C01796=1071.696,311.652,-94.387,174.617,30.497,155.487
C01797=1071.686,311.264,-94.337,174.612,30.490,155.486
C01798=1071.676,310.875,-94.286,174.607,30.483,155.484
C01799=1071.666,310.487,-94.236,174.603,30.476,155.483
C01800=1071.656,310.099,-94.186,174.597,30.469,155.482
C01801=1071.650,309.851,-94.154,174.595,30.465,155.481
C01802=1071.644,309.604,-94.121,174.592,30.460,155.480
C01803=1071.638,309.356,-94.089,174.589,30.456,155.480
C01804=1071.632,309.108,-94.057,174.586,30.451,155.479
C01805=1071.626,308.860,-94.025,174.582,30.447,155.478
C01806=1071.619,308.612,-93.993,174.580,30.443,155.477
C01807=1071.613,308.365,-93.960,174.577,30.439,155.477
C01808=1071.608,308.117,-93.929,174.573,30.434,155.476
C01809=1071.602,307.869,-93.897,174.571,30.430,155.475
C01810=1071.596,307.621,-93.865,174.567,30.425,155.474
C01811=1071.589,307.374,-93.833,174.565,30.421,155.473
C01812=1071.583,307.126,-93.801,174.562,30.417,155.473
C01813=1071.577,306.878,-93.769,174.558,30.412,155.472
C01814=1071.571,306.630,-93.737,174.556,30.408,155.471
C01815=1071.564,306.382,-93.705,174.552,30.403,155.470
C01816=1071.559,306.135,-93.673,174.550,30.399,155.470
C01817=1071.553,305.887,-93.641,174.547,30.395,155.469
C01818=1071.547,305.638,-93.609,174.543,30.390,155.468
C01819=1071.540,305.390,-93.578,174.541,30.386,155.467
C01820=1071.535,305.143,-93.546,174.538,30.382,155.467
C01821=1071.529,304.895,-93.513,174.535,30.377,155.466
C01822=1071.523,304.647,-93.481,174.532,30.373,155.465
C01823=1071.516,304.400,-93.450,174.529,30.368,155.464
C01824=1071.510,304.152,-93.418,174.526,30.364,155.463
C01825=1071.503,303.847,-93.379,174.522,30.359,155.463
C01826=1071.496,303.543,-93.340,174.519,30.354,155.462
C01827=1071.488,303.240,-93.301,174.515,30.348,155.461
C01828=1071.481,302.936,-93.263,174.512,30.343,155.460
C01829=1071.475,302.687,-93.231,174.508,30.338,155.459
C01830=1071.469,302.439,-93.199,174.506,30.334,155.458
C01831=1071.463,302.192,-93.167,174.503,30.330,155.457
C01832=1071.457,301.944,-93.135,174.499,30.325,155.457
C01833=1071.452,301.696,-93.104,174.497,30.321,155.456
C01834=1071.445,301.448,-93.072,174.494,30.317,155.455
C01835=1071.440,301.201,-93.041,174.492,30.313,155.454
C01836=1071.434,300.952,-93.009,174.488,30.308,155.454
C01837=1071.427,300.704,-92.978,174.485,30.304,155.453
C01838=1071.422,300.457,-92.946,174.483,30.299,155.452
C01839=1071.416,300.208,-92.914,174.479,30.295,155.451
C01840=1071.410,299.961,-92.883,174.477,30.291,155.451
C01841=1071.404,299.713,-92.851,174.474,30.287,155.450
C01842=1071.399,299.465,-92.820,174.470,30.282,155.449
C01843=1071.392,299.217,-92.789,174.468,30.278,155.448
C01844=1071.387,298.969,-92.757,174.465,30.273,155.448
C01845=1071.380,298.721,-92.726,174.463,30.270,155.447
C01846=1071.375,298.473,-92.695,174.459,30.265,155.446
C01847=1071.369,298.225,-92.663,174.456,30.261,155.445
C01848=1071.363,297.978,-92.632,174.454,30.256,155.445
C01849=1071.357,297.729,-92.600,174.450,30.252,155.444
C01850=1071.352,297.482,-92.569,174.448,30.248,155.443
C01851=1071.345,297.234,-92.537,174.445,30.243,155.442
C01852=1071.339,296.986,-92.507,174.442,30.239,155.442
C01853=1071.333,296.738,-92.475,174.439,30.235,155.441
C01854=1071.327,296.490,-92.444,174.436,30.231,155.440
C01855=1071.321,296.242,-92.412,174.434,30.226,155.439
C01856=1071.316,295.994,-92.382,174.431,30.222,155.439
C01857=1071.309,295.746,-92.351,174.427,30.218,155.438
C01858=1071.304,295.498,-92.319,174.425,30.214,155.437
C01859=1071.297,295.250,-92.288,174.422,30.210,155.436
C01860=1071.291,295.002,-92.258,174.420,30.205,155.436
C01861=1071.285,294.754,-92.227,174.416,30.201,155.435
C01862=1071.279,294.506,-92.196,174.414,30.197,155.434
C01863=1071.273,294.259,-92.165,174.411,30.193,155.434
C01864=1071.267,294.010,-92.134,174.408,30.189,155.433
C01865=1071.262,293.763,-92.102,174.405,30.184,155.432
C01866=1071.255,293.514,-92.071,174.402,30.180,155.431
C01867=1071.249,293.266,-92.041,174.400,30.176,155.431
C01868=1071.243,293.019,-92.010,174.397,30.172,155.430
C01869=1071.237,292.771,-91.979,174.393,30.167,155.429
C01870=1071.231,292.522,-91.948,174.391,30.164,155.429
C01871=1071.225,292.275,-91.917,174.388,30.159,155.428
C01872=1071.219,292.027,-91.887,174.386,30.155,155.427
C01873=1071.213,291.778,-91.856,174.382,30.151,155.426
C01874=1071.208,291.530,-91.825,174.379,30.147,155.426
C01875=1071.202,291.283,-91.794,174.377,30.143,155.425
C01876=1071.195,291.034,-91.763,174.374,30.139,155.424
C01877=1071.190,290.820,-91.736,174.372,30.135,155.424
C01878=1071.185,290.605,-91.709,174.369,30.131,155.423
C01879=1071.180,290.390,-91.684,174.366,30.128,155.422
C01880=1071.174,290.175,-91.657,174.365,30.124,155.422
C01881=1071.169,289.960,-91.630,174.362,30.120,155.421
C01882=1071.164,289.745,-91.603,174.359,30.117,155.420
C01883=1071.159,289.530,-91.577,174.357,30.113,155.420
C01884=1071.154,289.315,-91.551,174.355,30.109,155.419
C01885=1071.148,289.068,-91.520,174.352,30.105,155.419
C01886=1071.142,288.819,-91.489,174.349,30.101,155.418
C01887=1071.136,288.571,-91.459,174.346,30.097,155.417
C01888=1071.129,288.323,-91.428,174.344,30.093,155.416
C01889=1071.124,288.076,-91.397,174.341,30.089,155.416
C01890=1071.118,287.828,-91.367,174.338,30.085,155.415
C01891=1071.111,287.579,-91.336,174.335,30.080,155.414
C01892=1071.106,287.331,-91.306,174.332,30.077,155.414
C01893=1071.099,287.084,-91.276,174.330,30.073,155.413
C01894=1071.093,286.835,-91.245,174.327,30.068,155.412
C01895=1071.087,286.587,-91.216,174.324,30.064,155.411
C01896=1071.081,286.339,-91.185,174.321,30.060,155.411
C01897=1071.075,286.091,-91.155,174.318,30.056,155.410
C01898=1071.069,285.843,-91.124,174.316,30.052,155.409
C01899=1071.063,285.595,-91.094,174.313,30.048,155.409
C01900=1071.057,285.347,-91.064,174.311,30.044,155.408
C01901=1071.052,285.099,-91.033,174.307,30.040,155.407
C01902=1071.045,284.851,-91.003,174.305,30.035,155.407
C01903=1071.039,284.603,-90.972,174.302,30.032,155.406
C01904=1071.034,284.354,-90.943,174.299,30.027,155.405
C01905=1071.028,284.107,-90.912,174.297,30.023,155.404
C01906=1071.022,283.858,-90.882,174.294,30.019,155.404
C01907=1071.015,283.611,-90.852,174.291,30.015,155.403
C01908=1071.009,283.363,-90.821,174.288,30.011,155.402
C01909=1071.004,283.114,-90.792,174.286,30.007,155.402
C01910=1070.998,282.867,-90.761,174.283,30.003,155.401
C01911=1070.991,282.618,-90.731,174.280,29.999,155.400
C01912=1070.986,282.370,-90.701,174.278,29.994,155.399
C01913=1070.980,282.122,-90.671,174.275,29.991,155.399
C01914=1070.974,281.874,-90.640,174.272,29.986,155.398
C01915=1070.969,281.625,-90.611,174.269,29.982,155.397
C01916=1070.962,281.378,-90.581,174.266,29.978,155.397
C01917=1070.956,281.129,-90.550,174.264,29.974,155.396
C01918=1070.950,280.881,-90.521,174.261,29.970,155.395
C01919=1070.945,280.633,-90.490,174.259,29.966,155.395
C01920=1070.939,280.385,-90.460,174.256,29.962,155.394
C01921=1070.932,280.137,-90.431,174.254,29.958,155.393
C01922=1070.927,279.889,-90.401,174.251,29.954,155.393
C01923=1070.921,279.641,-90.371,174.248,29.949,155.392
C01924=1070.914,279.393,-90.341,174.245,29.945,155.391
C01925=1070.908,279.144,-90.311,174.242,29.942,155.391
C01926=1070.903,278.896,-90.281,174.240,29.937,155.390
C01927=1070.896,278.648,-90.252,174.237,29.933,155.389
C01928=1070.891,278.401,-90.221,174.235,29.929,155.388
C01929=1070.885,278.152,-90.192,174.232,29.926,155.388
C01930=1070.879,277.904,-90.163,174.229,29.921,155.387
C01931=1070.873,277.656,-90.132,174.227,29.917,155.386
C01932=1070.867,277.408,-90.103,174.223,29.913,155.386
C01933=1070.857,276.988,-90.052,174.219,29.906,155.384
C01934=1070.846,276.569,-90.002,174.215,29.899,155.383
C01935=1070.836,276.149,-89.952,174.210,29.893,155.382
C01936=1070.826,275.729,-89.902,174.206,29.886,155.381
C01937=1070.821,275.481,-89.872,174.204,29.882,155.380
C01938=1070.814,275.233,-89.843,174.200,29.878,155.380
C01939=1070.809,274.985,-89.813,174.198,29.873,155.379
C01940=1070.803,274.737,-89.784,174.195,29.869,155.378
C01941=1070.797,274.489,-89.754,174.192,29.866,155.378
C01942=1070.790,274.241,-89.725,174.190,29.862,155.377
C01943=1070.785,273.992,-89.695,174.187,29.857,155.376
C01944=1070.779,273.744,-89.666,174.185,29.853,155.376
C01945=1070.773,273.496,-89.636,174.182,29.849,155.375
C01946=1070.768,273.247,-89.607,174.180,29.846,155.374
C01947=1070.761,273.000,-89.577,174.177,29.841,155.373
C01948=1070.755,272.752,-89.548,174.174,29.837,155.373
C01949=1070.749,272.503,-89.518,174.172,29.833,155.372
C01950=1070.743,272.255,-89.489,174.169,29.829,155.371
C01951=1070.738,272.007,-89.459,174.167,29.826,155.371
C01952=1070.731,271.758,-89.430,174.164,29.821,155.370
C01953=1070.725,271.510,-89.401,174.162,29.817,155.369
C01954=1070.720,271.262,-89.372,174.159,29.813,155.369
C01955=1070.713,271.014,-89.343,174.156,29.809,155.368
C01956=1070.708,270.765,-89.313,174.153,29.805,155.367
C01957=1070.702,270.517,-89.284,174.150,29.801,155.367
C01958=1070.696,270.270,-89.255,174.148,29.797,155.366
C01959=1070.690,270.021,-89.226,174.145,29.793,155.365
C01960=1070.684,269.773,-89.197,174.143,29.789,155.365
C01961=1070.678,269.525,-89.168,174.140,29.785,155.364
C01962=1070.672,269.277,-89.138,174.138,29.781,155.363
C01963=1070.666,269.028,-89.109,174.135,29.777,155.363
C01964=1070.660,268.780,-89.080,174.132,29.773,155.362
C01965=1070.654,268.532,-89.050,174.130,29.769,155.361
C01966=1070.648,268.284,-89.021,174.127,29.765,155.361
C01967=1070.642,268.035,-88.993,174.125,29.761,155.360
C01968=1070.636,267.787,-88.964,174.122,29.757,155.359
C01969=1070.630,267.539,-88.935,174.120,29.753,155.359
C01970=1070.625,267.291,-88.906,174.117,29.749,155.358
C01971=1070.619,267.043,-88.877,174.115,29.745,155.357
C01972=1070.613,266.794,-88.848,174.112,29.741,155.357
C01973=1070.606,266.546,-88.819,174.109,29.738,155.356
C01974=1070.601,266.297,-88.790,174.107,29.733,155.355
C01975=1070.595,266.049,-88.761,174.104,29.729,155.355
C01976=1070.589,265.801,-88.732,174.102,29.725,155.354
C01977=1070.583,265.553,-88.704,174.099,29.721,155.353
C01978=1070.577,265.305,-88.674,174.097,29.717,155.353
C01979=1070.571,265.057,-88.645,174.094,29.713,155.352
C01980=1070.565,264.808,-88.617,174.092,29.709,155.351
C01981=1070.559,264.560,-88.587,174.089,29.705,155.351
C01982=1070.553,264.312,-88.558,174.087,29.701,155.350
C01983=1070.547,264.064,-88.530,174.084,29.697,155.349
C01984=1070.541,263.815,-88.501,174.081,29.694,155.349
C01985=1070.531,263.399,-88.453,174.077,29.686,155.347
C01986=1070.521,262.982,-88.406,174.073,29.680,155.346
C01987=1070.511,262.566,-88.357,174.069,29.673,155.345
C01988=1070.501,262.150,-88.309,174.064,29.667,155.344
C01989=1070.495,261.901,-88.281,174.062,29.663,155.343
C01990=1070.489,261.654,-88.252,174.059,29.659,155.343
C01991=1070.483,261.405,-88.224,174.057,29.655,155.342
C01992=1070.477,261.157,-88.195,174.054,29.651,155.342
C01993=1070.470,260.909,-88.167,174.052,29.647,155.341
C01994=1070.464,260.661,-88.138,174.049,29.643,155.340
C01995=1070.458,260.412,-88.110,174.047,29.640,155.340
C01996=1070.453,260.164,-88.082,174.044,29.636,155.339
C01997=1070.446,259.916,-88.053,174.042,29.632,155.338
C01998=1070.440,259.667,-88.025,174.040,29.628,155.338
C01999=1070.434,259.419,-87.996,174.037,29.624,155.337
C02000=1070.428,259.171,-87.968,174.035,29.620,155.336
C02001=1070.422,258.922,-87.940,174.032,29.616,155.336
C02002=1070.416,258.674,-87.911,174.030,29.612,155.335
C02003=1070.410,258.425,-87.883,174.027,29.608,155.334
C02004=1070.405,258.177,-87.855,174.025,29.604,155.334
C02005=1070.399,257.929,-87.826,174.022,29.601,155.333
C02006=1070.392,257.681,-87.798,174.019,29.597,155.332
C02007=1070.386,257.433,-87.770,174.017,29.592,155.332
C02008=1070.380,257.184,-87.741,174.014,29.588,155.331
C02009=1070.374,256.935,-87.713,174.012,29.584,155.330
C02010=1070.369,256.688,-87.684,174.009,29.580,155.330
C02011=1070.362,256.439,-87.657,174.007,29.576,155.329
C02012=1070.356,256.191,-87.628,174.004,29.573,155.328
C02013=1070.351,255.943,-87.600,174.003,29.569,155.328
C02014=1070.345,255.694,-87.572,174.000,29.565,155.327
C02015=1070.339,255.445,-87.544,173.998,29.561,155.326
C02016=1070.333,255.198,-87.516,173.995,29.557,155.326
C02017=1070.327,254.949,-87.487,173.993,29.553,155.325
C02018=1070.321,254.700,-87.459,173.990,29.549,155.325
C02019=1070.315,254.452,-87.431,173.988,29.545,155.324
C02020=1070.309,254.204,-87.403,173.985,29.541,155.323
C02021=1070.303,253.956,-87.375,173.982,29.537,155.322
C02022=1070.297,253.707,-87.347,173.980,29.533,155.322
C02023=1070.291,253.458,-87.319,173.978,29.529,155.321
C02024=1070.285,253.211,-87.291,173.976,29.525,155.320
C02025=1070.279,252.962,-87.263,173.973,29.521,155.320
C02026=1070.274,252.714,-87.235,173.971,29.517,155.319
C02027=1070.268,252.465,-87.207,173.968,29.513,155.318
C02028=1070.261,252.217,-87.179,173.966,29.509,155.318
C02029=1070.256,251.969,-87.151,173.963,29.505,155.317
C02030=1070.250,251.720,-87.123,173.961,29.501,155.316
C02031=1070.245,251.472,-87.095,173.958,29.497,155.316
C02032=1070.238,251.223,-87.067,173.957,29.494,155.315
C02033=1070.233,250.975,-87.039,173.954,29.490,155.315
C02034=1070.227,250.726,-87.011,173.952,29.485,155.314
C02035=1070.221,250.478,-86.983,173.949,29.481,155.313
C02036=1070.215,250.229,-86.956,173.947,29.477,155.312
C02037=1070.205,249.811,-86.909,173.942,29.471,155.311
C02038=1070.196,249.392,-86.862,173.938,29.464,155.310
C02039=1070.186,248.974,-86.815,173.935,29.457,155.309
C02040=1070.176,248.555,-86.768,173.931,29.451,155.308
C02041=1070.170,248.307,-86.740,173.928,29.446,155.307
C02042=1070.165,248.059,-86.712,173.926,29.442,155.307
C02043=1070.159,247.810,-86.685,173.923,29.438,155.306
C02044=1070.153,247.562,-86.657,173.921,29.434,155.305
C02045=1070.147,247.313,-86.629,173.919,29.431,155.305
C02046=1070.142,247.065,-86.602,173.917,29.426,155.304
C02047=1070.135,246.816,-86.574,173.914,29.422,155.303
C02048=1070.130,246.568,-86.546,173.912,29.418,155.303
C02049=1070.124,246.320,-86.519,173.909,29.414,155.302
C02050=1070.118,246.071,-86.491,173.907,29.410,155.301
C02051=1070.112,245.823,-86.464,173.905,29.407,155.301
C02052=1070.107,245.574,-86.436,173.902,29.403,155.300
C02053=1070.101,245.326,-86.409,173.900,29.399,155.299
C02054=1070.094,245.078,-86.381,173.897,29.395,155.299
C02055=1070.089,244.829,-86.354,173.895,29.390,155.298
C02056=1070.083,244.581,-86.326,173.892,29.386,155.297
C02057=1070.077,244.332,-86.299,173.891,29.383,155.297
C02058=1070.071,244.084,-86.271,173.888,29.379,155.296
C02059=1070.065,243.835,-86.244,173.886,29.375,155.295
C02060=1070.059,243.587,-86.216,173.883,29.371,155.295
C02061=1070.054,243.339,-86.189,173.881,29.367,155.294
C02062=1070.048,243.090,-86.161,173.879,29.363,155.293
C02063=1070.042,242.842,-86.135,173.877,29.359,155.293
C02064=1070.037,242.594,-86.107,173.874,29.355,155.292
C02065=1070.030,242.345,-86.080,173.872,29.351,155.291
C02066=1070.024,242.097,-86.052,173.869,29.347,155.291
C02067=1070.018,241.847,-86.025,173.868,29.343,155.290
C02068=1070.013,241.599,-85.998,173.865,29.339,155.289
C02069=1070.006,241.351,-85.970,173.863,29.335,155.289
C02070=1070.000,241.102,-85.944,173.860,29.331,155.288
C02071=1069.994,240.854,-85.917,173.858,29.327,155.287
C02072=1069.989,240.605,-85.889,173.856,29.324,155.287
C02073=1069.983,240.357,-85.862,173.854,29.320,155.286
C02074=1069.977,240.108,-85.836,173.851,29.316,155.285
C02075=1069.970,239.860,-85.808,173.849,29.312,155.285
C02076=1069.965,239.611,-85.781,173.846,29.308,155.284
C02077=1069.959,239.363,-85.754,173.845,29.304,155.284
C02078=1069.953,239.115,-85.726,173.842,29.300,155.283
C02079=1069.947,238.866,-85.700,173.840,29.296,155.282
C02080=1069.941,238.618,-85.673,173.837,29.292,155.281
C02081=1069.935,238.369,-85.646,173.835,29.288,155.281
C02082=1069.930,238.120,-85.619,173.833,29.284,155.280
C02083=1069.924,237.872,-85.591,173.831,29.280,155.280
C02084=1069.917,237.623,-85.564,173.828,29.276,155.279
C02085=1069.912,237.375,-85.538,173.826,29.272,155.278
C02086=1069.906,237.127,-85.511,173.824,29.268,155.278
C02087=1069.900,236.878,-85.484,173.822,29.264,155.277
C02088=1069.894,236.629,-85.457,173.819,29.260,155.276
C02089=1069.889,236.417,-85.434,173.818,29.257,155.276
C02090=1069.884,236.205,-85.411,173.815,29.253,155.275
C02091=1069.879,235.992,-85.388,173.813,29.250,155.275
C02092=1069.875,235.780,-85.365,173.812,29.247,155.274
C02093=1069.869,235.567,-85.342,173.809,29.243,155.273
C02094=1069.864,235.354,-85.319,173.808,29.240,155.273
C02095=1069.859,235.142,-85.296,173.806,29.236,155.272
C02096=1069.854,234.929,-85.273,173.804,29.233,155.272
C02097=1069.848,234.681,-85.246,173.801,29.229,155.271
C02098=1069.842,234.432,-85.219,173.800,29.225,155.270
C02099=1069.836,234.184,-85.192,173.797,29.221,155.270
C02100=1069.830,233.936,-85.166,173.795,29.217,155.269
C02101=1069.824,233.687,-85.139,173.792,29.213,155.268
C02102=1069.819,233.439,-85.112,173.791,29.209,155.268
C02103=1069.813,233.189,-85.086,173.788,29.205,155.267
C02104=1069.807,232.941,-85.060,173.786,29.201,155.266
C02105=1069.801,232.693,-85.033,173.783,29.197,155.266
C02106=1069.795,232.444,-85.006,173.782,29.193,155.265
C02107=1069.790,232.196,-84.980,173.779,29.189,155.265
C02108=1069.783,231.947,-84.953,173.777,29.185,155.264
C02109=1069.777,231.698,-84.926,173.775,29.181,155.263
C02110=1069.772,231.450,-84.899,173.773,29.177,155.262
C02111=1069.766,231.202,-84.873,173.770,29.173,155.262
C02112=1069.760,230.953,-84.846,173.768,29.169,155.261
C02113=1069.755,230.704,-84.820,173.766,29.166,155.260
C02114=1069.749,230.456,-84.793,173.764,29.162,155.260
C02115=1069.743,230.208,-84.767,173.761,29.158,155.259
C02116=1069.737,229.959,-84.740,173.760,29.154,155.259
C02117=1069.730,229.711,-84.714,173.757,29.149,155.258
C02118=1069.725,229.462,-84.688,173.755,29.145,155.257
C02119=1069.719,229.213,-84.661,173.752,29.141,155.257
C02120=1069.713,228.965,-84.634,173.751,29.138,155.256
C02121=1069.707,228.717,-84.608,173.748,29.134,155.255
C02122=1069.701,228.467,-84.582,173.746,29.130,155.255
C02123=1069.695,228.219,-84.555,173.744,29.126,155.254
C02124=1069.689,227.970,-84.529,173.742,29.122,155.253
C02125=1069.683,227.722,-84.503,173.739,29.118,155.253
C02126=1069.677,227.473,-84.477,173.737,29.114,155.252
C02127=1069.671,227.225,-84.450,173.735,29.110,155.251
C02128=1069.666,226.976,-84.424,173.733,29.106,155.251
C02129=1069.659,226.728,-84.398,173.730,29.102,155.250
C02130=1069.654,226.480,-84.372,173.729,29.098,155.249
C02131=1069.647,226.230,-84.345,173.726,29.094,155.249
C02132=1069.642,225.982,-84.319,173.724,29.090,155.248
C02133=1069.635,225.733,-84.293,173.722,29.086,155.247
C02134=1069.630,225.485,-84.267,173.720,29.082,155.247
C02135=1069.624,225.236,-84.241,173.718,29.078,155.246
C02136=1069.618,224.988,-84.215,173.716,29.074,155.245
C02137=1069.612,224.739,-84.189,173.714,29.070,155.245
C02138=1069.606,224.490,-84.162,173.711,29.066,155.244
C02139=1069.600,224.242,-84.136,173.710,29.062,155.243
C02140=1069.595,223.993,-84.110,173.707,29.058,155.243
C02141=1069.589,223.744,-84.084,173.705,29.054,155.242
C02142=1069.583,223.496,-84.058,173.703,29.050,155.241
C02143=1069.577,223.247,-84.032,173.701,29.046,155.241
C02144=1069.571,222.999,-84.005,173.698,29.042,155.240
C02145=1069.566,222.783,-83.983,173.697,29.039,155.239
C02146=1069.561,222.566,-83.960,173.695,29.035,155.239
C02147=1069.556,222.350,-83.938,173.693,29.031,155.238
C02148=1069.551,222.132,-83.915,173.691,29.028,155.238
C02149=1069.546,221.916,-83.893,173.690,29.025,155.237
C02150=1069.541,221.699,-83.869,173.687,29.021,155.237
C02151=1069.536,221.483,-83.847,173.686,29.018,155.236
C02152=1069.531,221.266,-83.824,173.684,29.015,155.235
C02153=1069.525,221.017,-83.799,173.682,29.010,155.235
C02154=1069.519,220.768,-83.773,173.679,29.006,155.234
C02155=1069.513,220.520,-83.747,173.678,29.002,155.233
C02156=1069.507,220.271,-83.721,173.675,28.998,155.233
C02157=1069.501,220.023,-83.696,173.673,28.994,155.232
C02158=1069.494,219.775,-83.669,173.671,28.991,155.231
C02159=1069.489,219.526,-83.644,173.669,28.987,155.231
C02160=1069.483,219.277,-83.618,173.667,28.983,155.230
C02161=1069.477,219.028,-83.592,173.665,28.979,155.230
C02162=1069.471,218.780,-83.566,173.662,28.975,155.229
C02163=1069.465,218.531,-83.540,173.661,28.970,155.228
C02164=1069.459,218.282,-83.515,173.658,28.966,155.227
C02165=1069.453,218.034,-83.490,173.656,28.962,155.227
C02166=1069.448,217.785,-83.464,173.654,28.959,155.226
C02167=1069.441,217.537,-83.438,173.652,28.955,155.226
C02168=1069.436,217.288,-83.412,173.650,28.951,155.225
C02169=1069.430,217.040,-83.387,173.648,28.947,155.224
C02170=1069.424,216.791,-83.361,173.646,28.942,155.223
C02171=1069.418,216.542,-83.335,173.644,28.939,155.223
C02172=1069.412,216.293,-83.310,173.642,28.935,155.222
C02173=1069.406,216.044,-83.284,173.639,28.931,155.222
C02174=1069.401,215.796,-83.259,173.638,28.927,155.221
C02175=1069.395,215.548,-83.234,173.635,28.922,155.220
C02176=1069.389,215.299,-83.207,173.634,28.919,155.219
C02177=1069.383,215.051,-83.182,173.631,28.914,155.219
C02178=1069.377,214.802,-83.156,173.629,28.910,155.218
C02179=1069.371,214.553,-83.131,173.627,28.907,155.218
C02180=1069.365,214.305,-83.106,173.625,28.902,155.217
C02181=1069.360,214.056,-83.080,173.624,28.898,155.216
C02182=1069.354,213.808,-83.054,173.621,28.894,155.215
C02183=1069.348,213.559,-83.029,173.619,28.890,155.215
C02184=1069.342,213.310,-83.003,173.617,28.886,155.214
C02185=1069.336,213.062,-82.978,173.615,28.882,155.213
C02186=1069.330,212.813,-82.953,173.613,28.878,155.213
C02187=1069.325,212.564,-82.927,173.611,28.874,155.212
C02188=1069.319,212.315,-82.902,173.608,28.870,155.211
C02189=1069.313,212.066,-82.877,173.607,28.866,155.211
C02190=1069.306,211.818,-82.852,173.605,28.862,155.210
C02191=1069.301,211.570,-82.827,173.603,28.858,155.209
C02192=1069.295,211.321,-82.801,173.601,28.854,155.209
C02193=1069.289,211.072,-82.775,173.599,28.850,155.208
C02194=1069.283,210.823,-82.750,173.597,28.846,155.207
C02195=1069.277,210.575,-82.725,173.594,28.842,155.207
C02196=1069.271,210.326,-82.700,173.593,28.838,155.206
C02197=1069.265,210.077,-82.675,173.590,28.834,155.205
C02198=1069.260,209.828,-82.649,173.589,28.830,155.205
C02199=1069.254,209.580,-82.624,173.587,28.826,155.204
C02200=1069.248,209.332,-82.599,173.585,28.822,155.203
C02201=1069.243,209.117,-82.577,173.583,28.818,155.203
C02202=1069.237,208.903,-82.556,173.581,28.815,155.202
C02203=1069.232,208.688,-82.534,173.580,28.811,155.202
C02204=1069.228,208.474,-82.513,173.578,28.808,155.201
C02205=1069.223,208.259,-82.491,173.576,28.804,155.200
C02206=1069.218,208.046,-82.469,173.574,28.801,155.200
C02207=1069.212,207.831,-82.448,173.572,28.798,155.199
C02208=1069.207,207.616,-82.426,173.571,28.794,155.199
C02209=1069.183,206.573,-82.323,173.428,28.722,155.196
C02210=1069.177,206.324,-82.299,173.427,28.718,155.195
C02211=1069.171,206.076,-82.275,173.424,28.715,155.195
C02212=1069.166,205.827,-82.251,173.422,28.712,155.194
C02213=1069.160,205.578,-82.226,173.420,28.709,155.194
C02214=1069.155,205.329,-82.202,173.418,28.706,155.193
C02215=1069.148,205.080,-82.178,173.415,28.703,155.193
C02216=1069.143,204.832,-82.154,173.414,28.700,155.192
C02217=1069.138,204.583,-82.129,173.411,28.697,155.192
C02218=1069.132,204.334,-82.105,173.409,28.693,155.191
C02219=1069.126,204.086,-82.081,173.407,28.690,155.191
C02220=1069.120,203.837,-82.057,173.404,28.687,155.190
C02221=1069.115,203.588,-82.032,173.402,28.684,155.190
C02222=1069.109,203.339,-82.008,173.400,28.681,155.190
C02223=1069.103,203.091,-81.984,173.398,28.678,155.189
C02224=1069.097,202.842,-81.960,173.395,28.675,155.189
C02225=1069.092,202.593,-81.935,173.394,28.672,155.188
C02226=1069.087,202.344,-81.911,173.391,28.669,155.188
C02227=1069.080,202.095,-81.887,173.389,28.665,155.187
C02228=1069.075,201.847,-81.863,173.387,28.662,155.187
C02229=1069.069,201.598,-81.840,173.384,28.660,155.187
C02230=1069.063,201.349,-81.815,173.382,28.656,155.186
C02231=1069.057,201.100,-81.792,173.380,28.653,155.186
C02232=1069.052,200.852,-81.767,173.378,28.650,155.185
C02233=1069.045,200.603,-81.743,173.376,28.647,155.185
C02234=1069.040,200.354,-81.719,173.374,28.644,155.184
C02235=1069.034,200.105,-81.696,173.371,28.641,155.184
C02236=1069.028,199.856,-81.672,173.370,28.638,155.183
C02237=1069.022,199.608,-81.648,173.367,28.635,155.183
C02238=1069.017,199.359,-81.624,173.364,28.632,155.183
C02239=1069.011,199.110,-81.600,173.363,28.629,155.182
C02240=1069.005,198.861,-81.577,173.360,28.626,155.182
C02241=1068.999,198.613,-81.552,173.359,28.623,155.181
C02242=1068.993,198.364,-81.528,173.356,28.620,155.181
C02243=1068.988,198.115,-81.505,173.354,28.617,155.180
C02244=1068.982,197.866,-81.481,173.352,28.614,155.180
C02245=1068.976,197.618,-81.457,173.350,28.611,155.180
C02246=1068.970,197.368,-81.434,173.348,28.608,155.179
C02247=1068.965,197.119,-81.409,173.345,28.605,155.179
C02248=1068.959,196.871,-81.386,173.343,28.602,155.178
C02249=1068.952,196.622,-81.362,173.341,28.599,155.178
C02250=1068.947,196.373,-81.338,173.339,28.596,155.177
C02251=1068.941,196.125,-81.315,173.337,28.593,155.177
C02252=1068.936,195.876,-81.291,173.335,28.590,155.177
C02253=1068.930,195.627,-81.267,173.332,28.587,155.176
C02254=1068.924,195.378,-81.243,173.331,28.584,155.176
C02255=1068.918,195.129,-81.220,173.328,28.581,155.175
C02256=1068.912,194.881,-81.196,173.326,28.578,155.175
C02257=1068.907,194.632,-81.173,173.324,28.575,155.174
C02258=1068.901,194.383,-81.149,173.322,28.572,155.174
C02259=1068.896,194.133,-81.125,173.320,28.569,155.173
C02260=1068.890,193.885,-81.101,173.317,28.566,155.173
C02261=1068.884,193.636,-81.078,173.316,28.563,155.173
C02262=1068.879,193.388,-81.054,173.313,28.560,155.172
C02263=1068.873,193.139,-81.031,173.312,28.557,155.172
C02264=1068.868,192.890,-81.007,173.309,28.554,155.171
C02265=1068.861,192.641,-80.984,173.307,28.551,155.171
C02266=1068.855,192.392,-80.960,173.305,28.548,155.170
C02267=1068.850,192.143,-80.936,173.303,28.545,155.170
C02268=1068.844,191.895,-80.913,173.301,28.542,155.170
C02269=1068.838,191.646,-80.890,173.298,28.538,155.169
C02270=1068.832,191.363,-80.862,173.297,28.536,155.169
C02271=1068.826,191.081,-80.836,173.294,28.532,155.168
C02272=1068.819,190.799,-80.809,173.292,28.529,155.168
C02273=1068.813,190.517,-80.783,173.289,28.525,155.167
C02274=1068.808,190.268,-80.759,173.287,28.522,155.167
C02275=1068.802,190.020,-80.736,173.285,28.519,155.166
C02276=1068.796,189.771,-80.713,173.283,28.516,155.166
C02277=1068.791,189.521,-80.689,173.281,28.513,155.165
C02278=1068.785,189.273,-80.666,173.279,28.510,155.165
C02279=1068.779,189.024,-80.643,173.277,28.507,155.165
C02280=1068.774,188.775,-80.619,173.274,28.504,155.164
C02281=1068.768,188.526,-80.595,173.273,28.501,155.164
C02282=1068.762,188.277,-80.572,173.270,28.498,155.163
C02283=1068.757,188.028,-80.549,173.269,28.495,155.163
C02284=1068.751,187.779,-80.526,173.266,28.492,155.162
C02285=1068.745,187.531,-80.502,173.265,28.489,155.162
C02286=1068.739,187.282,-80.479,173.262,28.486,155.161
C02287=1068.734,187.033,-80.456,173.261,28.483,155.161
C02288=1068.729,186.784,-80.433,173.258,28.480,155.161
C02289=1068.723,186.536,-80.409,173.257,28.477,155.160
C02290=1068.718,186.286,-80.385,173.254,28.474,155.160
C02291=1068.712,186.037,-80.362,173.252,28.471,155.159
C02292=1068.706,185.789,-80.339,173.250,28.468,155.159
C02293=1068.700,185.540,-80.317,173.248,28.465,155.158
C02294=1068.695,185.291,-80.292,173.246,28.462,155.158
C02295=1068.689,185.042,-80.269,173.244,28.459,155.158
C02296=1068.684,184.793,-80.246,173.242,28.456,155.157
C02297=1068.678,184.544,-80.223,173.240,28.453,155.157
C02298=1068.672,184.295,-80.200,173.238,28.450,155.156
C02299=1068.666,184.047,-80.178,173.236,28.448,155.156
C02300=1068.661,183.798,-80.155,173.233,28.445,155.156
C02301=1068.655,183.549,-80.132,173.232,28.442,155.155
C02302=1068.649,183.300,-80.109,173.229,28.439,155.155
C02303=1068.644,183.051,-80.086,173.228,28.436,155.154
C02304=1068.637,182.802,-80.063,173.225,28.433,155.154
C02305=1068.631,182.554,-80.040,173.224,28.430,155.153
C02306=1068.626,182.305,-80.018,173.221,28.427,155.153
C02307=1068.620,182.056,-79.995,173.220,28.424,155.153
C02308=1068.614,181.807,-79.972,173.218,28.422,155.152
C02309=1068.608,181.558,-79.949,173.215,28.419,155.152
C02310=1068.602,181.309,-79.926,173.214,28.416,155.151
C02311=1068.596,181.060,-79.903,173.211,28.413,155.151
C02312=1068.591,180.812,-79.880,173.210,28.410,155.151
C02313=1068.585,180.563,-79.857,173.207,28.407,155.150
C02314=1068.579,180.314,-79.835,173.206,28.405,155.150
C02315=1068.573,180.065,-79.812,173.203,28.402,155.149
C02316=1068.567,179.816,-79.789,173.201,28.399,155.149
C02317=1068.561,179.567,-79.766,173.199,28.396,155.149
C02318=1068.556,179.318,-79.744,173.197,28.393,155.148
C02319=1068.550,179.069,-79.721,173.195,28.390,155.148
C02320=1068.544,178.820,-79.698,173.193,28.387,155.147
C02321=1068.538,178.571,-79.676,173.192,28.385,155.147
C02322=1068.532,178.323,-79.653,173.189,28.382,155.147
C02323=1068.526,178.074,-79.630,173.187,28.379,155.146
C02324=1068.521,177.825,-79.607,173.185,28.376,155.146
C02325=1068.515,177.575,-79.585,173.183,28.373,155.145
C02326=1068.509,177.327,-79.562,173.181,28.370,155.145
C02327=1068.503,177.078,-79.539,173.179,28.367,155.145
C02328=1068.497,176.829,-79.517,173.178,28.364,155.144
C02329=1068.492,176.579,-79.494,173.175,28.361,155.144
C02330=1068.485,176.331,-79.472,173.174,28.359,155.143
C02331=1068.480,176.082,-79.449,173.171,28.356,155.143
C02332=1068.474,175.834,-79.426,173.169,28.353,155.143
C02333=1068.469,175.584,-79.404,173.167,28.350,155.142
C02334=1068.462,175.301,-79.379,173.165,28.347,155.142
C02335=1068.456,175.019,-79.353,173.163,28.344,155.141
C02336=1068.449,174.736,-79.327,173.160,28.340,155.141
C02337=1068.442,174.454,-79.302,173.158,28.337,155.140
C02338=1068.437,174.205,-79.279,173.156,28.334,155.140
C02339=1068.431,173.956,-79.256,173.155,28.331,155.139
C02340=1068.425,173.707,-79.234,173.152,28.328,155.139
C02341=1068.420,173.459,-79.212,173.151,28.326,155.139
C02342=1068.414,173.210,-79.189,173.148,28.323,155.138
C02343=1068.408,172.960,-79.167,173.147,28.320,155.138
C02344=1068.402,172.712,-79.144,173.145,28.317,155.137
C02345=1068.397,172.462,-79.122,173.143,28.314,155.137
C02346=1068.391,172.213,-79.099,173.141,28.311,155.137
C02347=1068.385,171.965,-79.077,173.139,28.309,155.136
C02348=1068.380,171.716,-79.055,173.137,28.306,155.136
C02349=1068.374,171.467,-79.032,173.135,28.303,155.135
C02350=1068.368,171.217,-79.010,173.133,28.299,155.135
C02351=1068.363,170.970,-78.988,173.131,28.297,155.135
C02352=1068.357,170.720,-78.966,173.130,28.294,155.134
C02353=1068.351,170.471,-78.943,173.127,28.291,155.134
C02354=1068.345,170.222,-78.921,173.126,28.288,155.133
C02355=1068.339,169.973,-78.898,173.123,28.285,155.133
C02356=1068.335,169.724,-78.876,173.121,28.283,155.133
C02357=1068.328,169.476,-78.854,173.120,28.280,155.132
C02358=1068.323,169.226,-78.832,173.117,28.277,155.132
C02359=1068.318,168.978,-78.809,173.116,28.274,155.131
C02360=1068.311,168.729,-78.787,173.114,28.271,155.131
C02361=1068.306,168.480,-78.764,173.112,28.268,155.130
C02362=1068.300,168.230,-78.742,173.110,28.265,155.130
C02363=1068.294,167.982,-78.720,173.109,28.262,155.130
C02364=1068.289,167.733,-78.698,173.106,28.259,155.129
C02365=1068.284,167.483,-78.676,173.104,28.257,155.129
C02366=1068.278,167.235,-78.654,173.103,28.254,155.128
C02367=1068.272,166.986,-78.632,173.100,28.251,155.128
C02368=1068.267,166.737,-78.609,173.099,28.248,155.128
C02369=1068.260,166.488,-78.587,173.097,28.245,155.127
C02370=1068.256,166.239,-78.565,173.095,28.242,155.127
C02371=1068.250,165.990,-78.542,173.093,28.239,155.126
C02372=1068.244,165.742,-78.521,173.092,28.236,155.126
C02373=1068.239,165.492,-78.499,173.089,28.233,155.125
C02374=1068.233,165.243,-78.476,173.088,28.231,155.125
C02375=1068.228,164.995,-78.454,173.086,28.228,155.125
C02376=1068.222,164.745,-78.432,173.083,28.225,155.124
C02377=1068.216,164.497,-78.410,173.082,28.222,155.124
C02378=1068.211,164.248,-78.388,173.080,28.219,155.123
C02379=1068.205,163.998,-78.366,173.078,28.216,155.123
C02380=1068.199,163.749,-78.344,173.076,28.213,155.123
C02381=1068.194,163.501,-78.322,173.075,28.211,155.122
C02382=1068.188,163.252,-78.300,173.072,28.208,155.122
C02383=1068.183,163.003,-78.278,173.071,28.205,155.121
C02384=1068.178,162.753,-78.256,173.069,28.202,155.121
C02385=1068.171,162.505,-78.233,173.067,28.199,155.120
C02386=1068.166,162.256,-78.212,173.065,28.196,155.120
C02387=1068.160,162.007,-78.190,173.064,28.193,155.120
C02388=1068.155,161.758,-78.168,173.061,28.190,155.119
C02389=1068.150,161.508,-78.146,173.059,28.187,155.119
C02390=1068.144,161.260,-78.125,173.058,28.185,155.118
C02391=1068.139,161.011,-78.102,173.055,28.182,155.118
C02392=1068.133,160.762,-78.080,173.054,28.179,155.118
C02393=1068.127,160.513,-78.059,173.052,28.176,155.117
C02394=1068.121,160.264,-78.037,173.051,28.173,155.117
C02395=1068.115,160.015,-78.015,173.048,28.170,155.116
C02396=1068.110,159.766,-77.994,173.047,28.168,155.116
C02397=1068.104,159.517,-77.972,173.045,28.165,155.116
C02398=1068.097,159.234,-77.948,173.043,28.161,155.115
C02399=1068.091,158.950,-77.922,173.040,28.158,155.115
C02400=1068.085,158.668,-77.898,173.039,28.155,155.114
C02401=1068.078,158.385,-77.874,173.036,28.152,155.114
C02402=1068.072,158.136,-77.852,173.035,28.149,155.113
C02403=1068.066,157.887,-77.830,173.033,28.147,155.113
C02404=1068.061,157.638,-77.808,173.030,28.144,155.113
C02405=1068.055,157.389,-77.787,173.029,28.141,155.112
C02406=1068.049,157.140,-77.766,173.027,28.138,155.112
C02407=1068.043,156.891,-77.744,173.026,28.135,155.111
C02408=1068.038,156.642,-77.722,173.023,28.132,155.111
C02409=1068.032,156.393,-77.700,173.022,28.130,155.111
C02410=1068.026,156.144,-77.679,173.020,28.127,155.110
C02411=1068.020,155.895,-77.658,173.018,28.124,155.110
C02412=1068.015,155.646,-77.635,173.016,28.121,155.109
C02413=1068.009,155.397,-77.614,173.014,28.118,155.109
C02414=1068.003,155.148,-77.592,173.013,28.116,155.109
C02415=1067.998,154.899,-77.571,173.010,28.113,155.108
C02416=1067.992,154.650,-77.550,173.009,28.110,155.108
C02417=1067.986,154.402,-77.528,173.007,28.107,155.107
C02418=1067.980,154.152,-77.507,173.006,28.104,155.107
C02419=1067.974,153.903,-77.486,173.003,28.101,155.107
C02420=1067.969,153.654,-77.464,173.002,28.099,155.106
C02421=1067.963,153.405,-77.442,173.000,28.096,155.106
C02422=1067.957,153.156,-77.421,172.998,28.093,155.105
C02423=1067.951,152.907,-77.399,172.996,28.090,155.105
C02424=1067.946,152.658,-77.379,172.994,28.087,155.105
C02425=1067.940,152.409,-77.357,172.993,28.085,155.104
C02426=1067.934,152.160,-77.336,172.990,28.082,155.104
C02427=1067.928,151.911,-77.314,172.989,28.079,155.104
C02428=1067.923,151.662,-77.294,172.987,28.077,155.103
C02429=1067.917,151.413,-77.272,172.986,28.074,155.103
C02430=1067.912,151.164,-77.250,172.983,28.071,155.102
C02431=1067.906,150.914,-77.228,172.982,28.068,155.102
C02432=1067.900,150.665,-77.208,172.980,28.065,155.102
C02433=1067.894,150.416,-77.186,172.978,28.063,155.101
C02434=1067.889,150.168,-77.165,172.976,28.060,155.101
C02435=1067.883,149.919,-77.144,172.974,28.057,155.100
C02436=1067.877,149.669,-77.123,172.973,28.054,155.100
C02437=1067.872,149.421,-77.102,172.971,28.051,155.100
C02438=1067.866,149.172,-77.080,172.970,28.049,155.099
C02439=1067.860,148.923,-77.059,172.967,28.046,155.099
C02440=1067.854,148.673,-77.038,172.966,28.043,155.098
C02441=1067.849,148.424,-77.017,172.964,28.040,155.098
C02442=1067.843,148.175,-76.996,172.963,28.037,155.098
C02443=1067.837,147.926,-76.974,172.960,28.034,155.097
C02444=1067.831,147.677,-76.953,172.959,28.032,155.097
C02445=1067.826,147.428,-76.932,172.957,28.029,155.096
C02446=1067.820,147.179,-76.912,172.955,28.026,155.096
C02447=1067.814,146.930,-76.891,172.954,28.023,155.095
C02448=1067.808,146.682,-76.869,172.951,28.021,155.095
C02449=1067.802,146.432,-76.848,172.950,28.018,155.095
C02450=1067.797,146.183,-76.827,172.948,28.015,155.094
C02451=1067.791,145.933,-76.806,172.947,28.013,155.094
C02452=1067.785,145.685,-76.785,172.944,28.010,155.094
C02453=1067.779,145.435,-76.765,172.943,28.007,155.093
C02454=1067.773,145.187,-76.743,172.941,28.004,155.093
C02455=1067.768,144.938,-76.723,172.939,28.001,155.092
C02456=1067.762,144.689,-76.701,172.938,27.999,155.092
C02457=1067.756,144.439,-76.681,172.935,27.996,155.092
C02458=1067.750,144.190,-76.659,172.934,27.993,155.091
C02459=1067.744,143.941,-76.639,172.932,27.991,155.091
C02460=1067.739,143.693,-76.618,172.931,27.988,155.091
C02461=1067.733,143.443,-76.597,172.929,27.985,155.090
C02462=1067.727,143.160,-76.573,172.927,27.982,155.090
C02463=1067.719,142.877,-76.549,172.925,27.979,155.089
C02464=1067.713,142.594,-76.526,172.923,27.975,155.089
C02465=1067.707,142.310,-76.502,172.921,27.973,155.088
C02466=1067.701,142.061,-76.480,172.919,27.970,155.088
C02467=1067.696,141.812,-76.460,172.917,27.967,155.088
C02468=1067.689,141.563,-76.440,172.916,27.964,155.087
C02469=1067.684,141.314,-76.418,172.914,27.961,155.087
C02470=1067.678,141.065,-76.398,172.913,27.958,155.086
C02471=1067.673,140.815,-76.377,172.910,27.955,155.086
C02472=1067.667,140.567,-76.356,172.908,27.953,155.086
C02473=1067.661,140.318,-76.336,172.907,27.950,155.085
C02474=1067.655,140.068,-76.315,172.905,27.947,155.085
C02475=1067.650,139.820,-76.293,172.904,27.944,155.084
C02476=1067.644,139.571,-76.273,172.902,27.942,155.084
C02477=1067.638,139.321,-76.253,172.900,27.939,155.084
C02478=1067.632,139.073,-76.231,172.898,27.936,155.083
C02479=1067.626,138.824,-76.211,172.897,27.934,155.083
C02480=1067.620,138.574,-76.190,172.895,27.931,155.082
C02481=1067.615,138.325,-76.170,172.894,27.928,155.082
C02482=1067.609,138.077,-76.149,172.892,27.925,155.082
C02483=1067.604,137.828,-76.129,172.890,27.922,155.081
C02484=1067.598,137.578,-76.108,172.888,27.920,155.081
C02485=1067.592,137.329,-76.088,172.886,27.917,155.080
C02486=1067.586,137.080,-76.067,172.885,27.914,155.080
C02487=1067.580,136.831,-76.046,172.883,27.911,155.080
C02488=1067.574,136.582,-76.026,172.882,27.909,155.079
C02489=1067.568,136.333,-76.006,172.879,27.906,155.079
C02490=1067.562,136.083,-75.985,172.878,27.903,155.079
C02491=1067.557,135.834,-75.964,172.876,27.901,155.078
C02492=1067.551,135.585,-75.944,172.875,27.898,155.078
C02493=1067.546,135.337,-75.923,172.873,27.895,155.077
C02494=1067.539,135.087,-75.903,172.872,27.892,155.077
C02495=1067.534,134.838,-75.882,172.869,27.889,155.077
C02496=1067.528,134.589,-75.862,172.867,27.886,155.076
C02497=1067.522,134.340,-75.842,172.866,27.884,155.076
C02498=1067.517,134.090,-75.821,172.864,27.881,155.075
C02499=1067.511,133.841,-75.801,172.863,27.879,155.075
C02500=1067.505,133.592,-75.780,172.861,27.876,155.075
C02501=1067.499,133.344,-75.760,172.860,27.873,155.074
C02502=1067.494,133.094,-75.740,172.857,27.870,155.074
C02503=1067.487,132.846,-75.719,172.856,27.867,155.073
C02504=1067.482,132.596,-75.698,172.854,27.865,155.073
C02505=1067.476,132.348,-75.678,172.853,27.862,155.073
C02506=1067.471,132.098,-75.657,172.851,27.859,155.072
C02507=1067.464,131.849,-75.637,172.850,27.856,155.072
C02508=1067.459,131.600,-75.617,172.848,27.854,155.071
C02509=1067.453,131.351,-75.597,172.846,27.851,155.071
C02510=1067.447,131.102,-75.577,172.844,27.848,155.071
C02511=1067.441,130.852,-75.556,172.842,27.846,155.070
C02512=1067.435,130.603,-75.537,172.841,27.843,155.070
C02513=1067.429,130.354,-75.517,172.839,27.840,155.070
C02514=1067.424,130.105,-75.496,172.838,27.837,155.069
C02515=1067.418,129.855,-75.476,172.836,27.835,155.069
C02516=1067.412,129.607,-75.456,172.834,27.832,155.068
C02517=1067.406,129.358,-75.436,172.832,27.829,155.068
C02518=1067.400,129.109,-75.415,172.831,27.826,155.068
C02519=1067.394,128.860,-75.395,172.829,27.824,155.067
C02520=1067.388,128.610,-75.375,172.827,27.821,155.067
C02521=1067.382,128.361,-75.354,172.826,27.819,155.067
C02522=1067.377,128.112,-75.335,172.824,27.816,155.066
C02523=1067.371,127.863,-75.315,172.823,27.813,155.066
C02524=1067.365,127.614,-75.295,172.820,27.810,155.065
C02525=1067.359,127.364,-75.274,172.819,27.807,155.065
C02526=1067.352,127.081,-75.251,172.817,27.805,155.065
C02527=1067.345,126.798,-75.229,172.816,27.802,155.064
C02528=1067.339,126.515,-75.206,172.813,27.798,155.064
C02529=1067.332,126.231,-75.184,172.812,27.795,155.063
C02530=1067.326,125.982,-75.164,172.810,27.793,155.063
C02531=1067.321,125.733,-75.143,172.808,27.790,155.063
C02532=1067.315,125.484,-75.123,172.806,27.787,155.062
C02533=1067.309,125.235,-75.104,172.805,27.784,155.062
C02534=1067.303,124.985,-75.084,172.803,27.781,155.061
C02535=1067.297,124.737,-75.064,172.802,27.779,155.061
C02536=1067.291,124.487,-75.043,172.800,27.776,155.061
C02537=1067.286,124.238,-75.024,172.799,27.774,155.060
C02538=1067.280,123.989,-75.004,172.797,27.771,155.060
C02539=1067.274,123.740,-74.984,172.795,27.768,155.059
C02540=1067.269,123.491,-74.964,172.794,27.765,155.059
C02541=1067.263,123.242,-74.944,172.791,27.762,155.059
C02542=1067.257,122.993,-74.924,172.790,27.759,155.058
C02543=1067.251,122.744,-74.905,172.788,27.757,155.058
C02544=1067.244,122.494,-74.885,172.787,27.754,155.058
C02545=1067.239,122.245,-74.864,172.785,27.752,155.057
C02546=1067.233,121.995,-74.845,172.784,27.749,155.057
C02547=1067.227,121.747,-74.825,172.782,27.746,155.056
C02548=1067.221,121.498,-74.805,172.781,27.743,155.056
C02549=1067.216,121.248,-74.786,172.779,27.741,155.056
C02550=1067.211,120.999,-74.765,172.778,27.738,155.055
C02551=1067.205,120.750,-74.745,172.776,27.735,155.055
C02552=1067.199,120.501,-74.726,172.774,27.732,155.054
C02553=1067.193,120.252,-74.706,172.772,27.729,155.054
C02554=1067.187,120.003,-74.687,172.771,27.726,155.054
C02555=1067.182,119.754,-74.666,172.769,27.724,155.053
C02556=1067.176,119.504,-74.647,172.768,27.721,155.053
C02557=1067.170,119.255,-74.627,172.766,27.719,155.052
C02558=1067.164,119.007,-74.607,172.764,27.716,155.052
C02559=1067.159,118.757,-74.588,172.763,27.713,155.052
C02560=1067.153,118.508,-74.568,172.761,27.710,155.051
C02561=1067.148,118.259,-74.548,172.760,27.708,155.051
C02562=1067.142,118.010,-74.528,172.758,27.705,155.050
C02563=1067.136,117.760,-74.509,172.757,27.702,155.050
C02564=1067.130,117.512,-74.489,172.755,27.699,155.050
C02565=1067.124,117.262,-74.469,172.754,27.696,155.049
C02566=1067.118,117.013,-74.449,172.751,27.693,155.049
C02567=1067.113,116.764,-74.430,172.750,27.691,155.048
C02568=1067.107,116.515,-74.410,172.748,27.688,155.048
C02569=1067.102,116.265,-74.390,172.747,27.685,155.048
C02570=1067.096,116.016,-74.371,172.745,27.682,155.047
C02571=1067.090,115.767,-74.351,172.744,27.679,155.047
C02572=1067.084,115.518,-74.332,172.742,27.677,155.046
C02573=1067.078,115.269,-74.312,172.741,27.674,155.046
C02574=1067.073,115.019,-74.293,172.739,27.671,155.046
C02575=1067.067,114.770,-74.272,172.738,27.668,155.045
C02576=1067.062,114.522,-74.253,172.736,27.666,155.045
C02577=1067.057,114.272,-74.234,172.735,27.663,155.044
C02578=1067.051,114.023,-74.214,172.733,27.660,155.044
C02579=1067.045,113.774,-74.195,172.731,27.657,155.044
C02580=1067.039,113.524,-74.176,172.730,27.655,155.043
C02581=1067.033,113.276,-74.156,172.728,27.652,155.043
C02582=1067.027,113.027,-74.137,172.727,27.649,155.042
C02583=1067.021,112.777,-74.118,172.724,27.646,155.042
C02584=1067.015,112.528,-74.098,172.723,27.644,155.042
C02585=1067.009,112.279,-74.079,172.721,27.641,155.041
C02586=1067.004,112.029,-74.059,172.720,27.638,155.041
C02587=1066.998,111.781,-74.039,172.718,27.635,155.041
C02588=1066.992,111.531,-74.020,172.717,27.632,155.040
C02589=1066.986,111.282,-74.001,172.715,27.630,155.040
C02590=1066.979,110.998,-73.979,172.714,27.627,155.039
C02591=1066.973,110.715,-73.957,172.712,27.624,155.039
C02592=1066.967,110.432,-73.935,172.710,27.620,155.038
C02593=1066.959,110.148,-73.913,172.708,27.618,155.038
C02594=1066.954,109.899,-73.894,172.707,27.615,155.038
C02595=1066.948,109.650,-73.875,172.705,27.612,155.037
C02596=1066.941,109.400,-73.856,172.704,27.610,155.037
C02597=1066.936,109.151,-73.837,172.702,27.607,155.037
C02598=1066.930,108.902,-73.817,172.701,27.604,155.036
C02599=1066.924,108.653,-73.798,172.699,27.601,155.036
C02600=1066.919,108.404,-73.779,172.698,27.599,155.035
C02601=1066.913,108.155,-73.760,172.696,27.596,155.035
C02602=1066.907,107.905,-73.741,172.695,27.593,155.035
C02603=1066.901,107.656,-73.722,172.692,27.591,155.034
C02604=1066.895,107.407,-73.702,172.691,27.588,155.034
C02605=1066.889,107.158,-73.683,172.689,27.585,155.033
C02606=1066.883,106.909,-73.664,172.688,27.582,155.033
C02607=1066.877,106.659,-73.644,172.686,27.579,155.033
C02608=1066.871,106.410,-73.626,172.685,27.577,155.032
C02609=1066.866,106.161,-73.607,172.683,27.574,155.032
C02610=1066.860,105.912,-73.588,172.681,27.571,155.031
C02611=1066.854,105.663,-73.568,172.680,27.569,155.031
C02612=1066.848,105.413,-73.550,172.678,27.566,155.031
C02613=1066.842,105.164,-73.531,172.677,27.563,155.030
C02614=1066.837,104.915,-73.511,172.675,27.560,155.030
C02615=1066.831,104.665,-73.492,172.674,27.558,155.030
C02616=1066.825,104.417,-73.474,172.672,27.555,155.029
C02617=1066.819,104.167,-73.455,172.671,27.552,155.029
C02618=1066.814,103.918,-73.435,172.669,27.549,155.028
C02619=1066.807,103.669,-73.417,172.668,27.547,155.028
C02620=1066.802,103.419,-73.397,172.666,27.544,155.028
C02621=1066.797,103.171,-73.379,172.665,27.541,155.027
C02622=1066.791,102.921,-73.359,172.663,27.539,155.027
C02623=1066.784,102.672,-73.341,172.662,27.536,155.026
C02624=1066.779,102.423,-73.321,172.660,27.533,155.026
C02625=1066.773,102.173,-73.302,172.659,27.530,155.026
C02626=1066.767,101.925,-73.284,172.657,27.528,155.025
C02627=1066.762,101.675,-73.265,172.656,27.525,155.025
C02628=1066.756,101.426,-73.245,172.654,27.522,155.024
C02629=1066.749,101.177,-73.227,172.653,27.519,155.024
C02630=1066.744,100.928,-73.208,172.651,27.516,155.024
C02631=1066.738,100.679,-73.189,172.650,27.514,155.023
C02632=1066.732,100.429,-73.170,172.648,27.511,155.023
C02633=1066.726,100.180,-73.151,172.647,27.509,155.023
C02634=1066.720,99.930,-73.133,172.645,27.506,155.022
C02635=1066.714,99.681,-73.114,172.644,27.503,155.022
C02636=1066.709,99.432,-73.095,172.642,27.500,155.021
C02637=1066.703,99.183,-73.077,172.641,27.497,155.021
C02638=1066.697,98.934,-73.057,172.639,27.495,155.021
C02639=1066.690,98.685,-73.039,172.637,27.492,155.020
C02640=1066.686,98.435,-73.021,172.636,27.489,155.020
C02641=1066.679,98.186,-73.002,172.634,27.487,155.019
C02642=1066.674,97.937,-72.983,172.633,27.484,155.019
C02643=1066.667,97.688,-72.964,172.631,27.481,155.019
C02644=1066.661,97.438,-72.945,172.630,27.478,155.018
C02645=1066.656,97.189,-72.927,172.628,27.476,155.018
C02646=1066.650,96.940,-72.908,172.627,27.473,155.018
C02647=1066.644,96.691,-72.889,172.625,27.470,155.017
C02648=1066.637,96.442,-72.871,172.624,27.468,155.017
C02649=1066.633,96.192,-72.853,172.622,27.465,155.016
C02650=1066.626,95.943,-72.834,172.621,27.462,155.016
C02651=1066.620,95.694,-72.815,172.619,27.459,155.016
C02652=1066.615,95.445,-72.796,172.618,27.456,155.015
C02653=1066.609,95.195,-72.778,172.616,27.454,155.015
C02654=1066.602,94.912,-72.756,172.615,27.451,155.014
C02655=1066.596,94.629,-72.735,172.612,27.448,155.014
C02656=1066.589,94.345,-72.714,172.611,27.444,155.013
C02657=1066.582,94.062,-72.693,172.609,27.442,155.013
C02658=1066.577,93.812,-72.675,172.608,27.439,155.013
C02659=1066.571,93.564,-72.656,172.606,27.436,155.012
C02660=1066.564,93.314,-72.638,172.605,27.433,155.012
C02661=1066.559,93.064,-72.619,172.603,27.430,155.011
C02662=1066.553,92.816,-72.601,172.602,27.428,155.011
C02663=1066.548,92.566,-72.582,172.600,27.425,155.011
C02664=1066.541,92.317,-72.564,172.599,27.422,155.010
C02665=1066.535,92.068,-72.545,172.597,27.420,155.010
C02666=1066.530,91.818,-72.527,172.596,27.417,155.010
C02667=1066.524,91.569,-72.508,172.594,27.414,155.009
C02668=1066.519,91.320,-72.490,172.593,27.411,155.009
C02669=1066.512,91.071,-72.471,172.591,27.409,155.008
C02670=1066.506,90.822,-72.453,172.590,27.406,155.008
C02671=1066.501,90.572,-72.435,172.588,27.403,155.008
C02672=1066.495,90.323,-72.416,172.587,27.400,155.007
C02673=1066.489,90.073,-72.398,172.585,27.398,155.007
C02674=1066.483,89.825,-72.380,172.584,27.395,155.006
C02675=1066.477,89.575,-72.362,172.582,27.392,155.006
C02676=1066.471,89.326,-72.343,172.581,27.389,155.006
C02677=1066.466,89.077,-72.325,172.579,27.387,155.005
C02678=1066.459,88.828,-72.306,172.578,27.384,155.005
C02679=1066.453,88.578,-72.288,172.576,27.382,155.005
C02680=1066.447,88.329,-72.270,172.575,27.379,155.004
C02681=1066.441,88.080,-72.252,172.573,27.376,155.004
C02682=1066.436,87.830,-72.234,172.572,27.373,155.003
C02683=1066.430,87.581,-72.215,172.570,27.370,155.003
C02684=1066.424,87.331,-72.197,172.569,27.368,155.003
C02685=1066.417,87.082,-72.179,172.567,27.365,155.002
C02686=1066.412,86.833,-72.161,172.566,27.363,155.002
C02687=1066.405,86.584,-72.143,172.564,27.360,155.002
C02688=1066.401,86.335,-72.124,172.563,27.357,155.001
C02689=1066.394,86.085,-72.106,172.561,27.354,155.001
C02690=1066.388,85.836,-72.088,172.560,27.351,155.000
C02691=1066.382,85.587,-72.070,172.558,27.349,155.000
C02692=1066.376,85.338,-72.052,172.557,27.346,155.000
C02693=1066.371,85.089,-72.034,172.555,27.343,154.999
C02694=1066.364,84.839,-72.016,172.554,27.341,154.999
C02695=1066.359,84.590,-71.997,172.552,27.338,154.998
C02696=1066.353,84.341,-71.979,172.551,27.335,154.998
C02697=1066.347,84.091,-71.961,172.550,27.332,154.998
C02698=1066.341,83.842,-71.943,172.549,27.330,154.997
C02699=1066.335,83.593,-71.925,172.547,27.327,154.997
C02700=1066.330,83.344,-71.908,172.546,27.325,154.997
C02701=1066.323,83.094,-71.889,172.544,27.322,154.996
C02702=1066.318,82.845,-71.871,172.543,27.319,154.996
C02703=1066.312,82.596,-71.853,172.541,27.316,154.995
C02704=1066.306,82.346,-71.835,172.540,27.313,154.995
C02705=1066.300,82.097,-71.817,172.538,27.311,154.995
C02706=1066.294,81.847,-71.799,172.537,27.308,154.994
C02707=1066.289,81.598,-71.781,172.535,27.305,154.994
C02708=1066.283,81.349,-71.763,172.534,27.303,154.993
C02709=1066.277,81.100,-71.745,172.532,27.300,154.993
C02710=1066.271,80.851,-71.727,172.531,27.297,154.993
C02711=1066.265,80.602,-71.709,172.529,27.294,154.992
C02712=1066.259,80.352,-71.691,172.528,27.291,154.992
C02713=1066.253,80.103,-71.673,172.526,27.289,154.991
C02714=1066.247,79.854,-71.655,172.525,27.286,154.991
C02715=1066.242,79.604,-71.637,172.523,27.283,154.991
C02716=1066.236,79.355,-71.619,172.522,27.280,154.990
C02717=1066.231,79.105,-71.602,172.520,27.278,154.990
C02718=1066.224,78.823,-71.582,172.519,27.275,154.989
C02719=1066.217,78.539,-71.561,172.517,27.272,154.989
C02720=1066.210,78.255,-71.541,172.516,27.268,154.989
C02721=1066.203,77.972,-71.521,172.513,27.265,154.988
C02722=1066.198,77.723,-71.503,172.512,27.262,154.988
C02723=1066.192,77.473,-71.485,172.510,27.260,154.987
C02724=1066.186,77.225,-71.467,172.510,27.257,154.987
C02725=1066.180,76.975,-71.449,172.508,27.255,154.987
C02726=1066.174,76.726,-71.431,172.507,27.252,154.986
C02727=1066.167,76.476,-71.414,172.505,27.249,154.986
C02728=1066.162,76.227,-71.396,172.504,27.246,154.985
C02729=1066.156,75.978,-71.378,172.502,27.244,154.985
C02730=1066.150,75.729,-71.361,172.501,27.241,154.985
C02731=1066.144,75.479,-71.343,172.499,27.238,154.984
C02732=1066.139,75.230,-71.325,172.498,27.236,154.984
C02733=1066.132,74.980,-71.307,172.496,27.233,154.984
C02734=1066.126,74.731,-71.290,172.495,27.230,154.983
C02735=1066.120,74.482,-71.272,172.493,27.227,154.983
C02736=1066.115,74.232,-71.255,172.492,27.225,154.983
C02737=1066.109,73.983,-71.237,172.490,27.222,154.982
C02738=1066.103,73.734,-71.219,172.489,27.219,154.982
C02739=1066.097,73.485,-71.202,172.487,27.216,154.981
C02740=1066.091,73.235,-71.185,172.486,27.214,154.981
C02741=1066.085,72.986,-71.167,172.484,27.211,154.981
C02742=1066.079,72.736,-71.149,172.483,27.208,154.980
C02743=1066.073,72.487,-71.131,172.481,27.206,154.980
C02744=1066.068,72.238,-71.114,172.480,27.203,154.979
C02745=1066.062,71.989,-71.096,172.479,27.200,154.979
C02746=1066.056,71.740,-71.079,172.478,27.198,154.979
C02747=1066.049,71.490,-71.061,172.476,27.195,154.978
C02748=1066.044,71.241,-71.044,172.475,27.192,154.978
C02749=1066.039,70.991,-71.027,172.473,27.190,154.978
C02750=1066.032,70.742,-71.009,172.472,27.187,154.977
C02751=1066.026,70.493,-70.992,172.470,27.184,154.977
C02752=1066.020,70.243,-70.974,172.469,27.181,154.976
C02753=1066.015,69.994,-70.956,172.467,27.178,154.976
C02754=1066.009,69.745,-70.939,172.466,27.176,154.976
C02755=1066.002,69.496,-70.921,172.464,27.173,154.975
C02756=1065.997,69.246,-70.904,172.463,27.170,154.975
C02757=1065.991,68.996,-70.887,172.461,27.168,154.974
C02758=1065.985,68.748,-70.870,172.460,27.165,154.974
C02759=1065.979,68.499,-70.852,172.458,27.162,154.974
C02760=1065.973,68.249,-70.834,172.457,27.159,154.973
C02761=1065.967,67.999,-70.818,172.455,27.157,154.973
C02762=1065.962,67.750,-70.800,172.455,27.154,154.973
C02763=1065.955,67.501,-70.782,172.453,27.152,154.972
C02764=1065.949,67.252,-70.765,172.452,27.149,154.972
C02765=1065.943,67.002,-70.748,172.450,27.146,154.971
C02766=1065.937,66.753,-70.731,172.449,27.143,154.971
C02767=1065.932,66.504,-70.714,172.447,27.141,154.971
C02768=1065.925,66.254,-70.696,172.446,27.138,154.970
C02769=1065.920,66.005,-70.679,172.445,27.135,154.970
C02770=1065.914,65.756,-70.662,172.443,27.132,154.970
C02771=1065.908,65.506,-70.644,172.442,27.130,154.969
C02772=1065.902,65.257,-70.627,172.440,27.127,154.969
C02773=1065.896,65.008,-70.610,172.439,27.124,154.968
C02774=1065.890,64.758,-70.593,172.437,27.122,154.968
C02775=1065.884,64.509,-70.575,172.436,27.119,154.968
C02776=1065.878,64.260,-70.559,172.434,27.116,154.967
C02777=1065.872,64.010,-70.541,172.433,27.114,154.967
C02778=1065.866,63.761,-70.524,172.431,27.111,154.967
C02779=1065.860,63.511,-70.507,172.431,27.108,154.966
C02780=1065.854,63.262,-70.490,172.429,27.106,154.966
C02781=1065.848,63.013,-70.474,172.428,27.103,154.965
C02782=1065.841,62.730,-70.453,172.425,27.100,154.965
C02783=1065.834,62.446,-70.434,172.424,27.097,154.965
C02784=1065.827,62.163,-70.415,172.422,27.094,154.964
C02785=1065.820,61.879,-70.395,172.421,27.091,154.964
C02786=1065.814,61.629,-70.378,172.419,27.088,154.963
C02787=1065.808,61.380,-70.361,172.418,27.085,154.963
C02788=1065.802,61.131,-70.344,172.416,27.083,154.963
C02789=1065.796,60.881,-70.327,172.415,27.080,154.962
C02790=1065.790,60.632,-70.310,172.413,27.077,154.962
C02791=1065.784,60.383,-70.294,172.412,27.075,154.962
C02792=1065.778,60.133,-70.276,172.410,27.072,154.961
C02793=1065.772,59.884,-70.260,172.409,27.070,154.961
C02794=1065.765,59.635,-70.243,172.407,27.067,154.960
C02795=1065.760,59.385,-70.225,172.406,27.064,154.960
C02796=1065.753,59.136,-70.209,172.405,27.062,154.960
C02797=1065.748,58.886,-70.192,172.404,27.059,154.959
C02798=1065.742,58.638,-70.175,172.402,27.056,154.959
C02799=1065.735,58.388,-70.158,172.401,27.054,154.959
C02800=1065.730,58.139,-70.141,172.399,27.051,154.958
C02801=1065.724,57.889,-70.124,172.398,27.048,154.958
C02802=1065.717,57.640,-70.107,172.396,27.045,154.958
C02803=1065.712,57.390,-70.090,172.395,27.043,154.957
C02804=1065.706,57.141,-70.074,172.393,27.040,154.957
C02805=1065.700,56.892,-70.057,172.392,27.038,154.956
C02806=1065.694,56.642,-70.040,172.390,27.035,154.956
C02807=1065.688,56.393,-70.023,172.389,27.032,154.956
C02808=1065.682,56.144,-70.006,172.387,27.030,154.955
C02809=1065.676,55.894,-69.990,172.386,27.027,154.955
C02810=1065.670,55.645,-69.973,172.384,27.024,154.955
C02811=1065.664,55.395,-69.956,172.384,27.022,154.954
C02812=1065.657,55.146,-69.939,172.382,27.019,154.954
C02813=1065.652,54.897,-69.922,172.381,27.016,154.953
C02814=1065.646,54.647,-69.906,172.379,27.013,154.953
C02815=1065.640,54.399,-69.889,172.378,27.011,154.953
C02816=1065.634,54.148,-69.872,172.376,27.008,154.952
C02817=1065.628,53.899,-69.855,172.375,27.006,154.952
C02818=1065.622,53.650,-69.838,172.374,27.003,154.952
C02819=1065.616,53.401,-69.822,172.372,27.000,154.951
C02820=1065.611,53.151,-69.805,172.371,26.998,154.951
C02821=1065.604,52.902,-69.788,172.369,26.995,154.951
C02822=1065.598,52.652,-69.772,172.368,26.992,154.950
C02823=1065.593,52.403,-69.755,172.366,26.989,154.950
C02824=1065.587,52.153,-69.739,172.365,26.987,154.949
C02825=1065.580,51.905,-69.722,172.364,26.984,154.949
C02826=1065.575,51.655,-69.705,172.363,26.981,154.949
C02827=1065.569,51.405,-69.688,172.361,26.979,154.948
C02828=1065.562,51.156,-69.671,172.360,26.976,154.948
C02829=1065.557,50.907,-69.655,172.358,26.973,154.948
C02830=1065.551,50.658,-69.639,172.357,26.971,154.947
C02831=1065.545,50.408,-69.622,172.355,26.968,154.947
C02832=1065.539,50.159,-69.606,172.354,26.965,154.946
C02833=1065.533,49.910,-69.589,172.352,26.962,154.946
C02834=1065.527,49.661,-69.572,172.351,26.960,154.946
C02835=1065.521,49.410,-69.555,172.349,26.957,154.945
C02836=1065.515,49.161,-69.539,172.348,26.954,154.945
C02837=1065.509,48.911,-69.523,172.346,26.951,154.945
C02838=1065.503,48.663,-69.506,172.346,26.949,154.944
C02839=1065.498,48.413,-69.489,172.344,26.946,154.944
C02840=1065.492,48.164,-69.473,172.343,26.944,154.943
C02841=1065.486,47.914,-69.456,172.341,26.941,154.943
C02842=1065.480,47.665,-69.440,172.340,26.938,154.943
C02843=1065.475,47.415,-69.423,172.338,26.935,154.942
C02844=1065.469,47.166,-69.407,172.337,26.933,154.942
C02845=1065.463,46.917,-69.390,172.335,26.930,154.942
C02846=1065.456,46.633,-69.371,172.334,26.927,154.941
C02847=1065.450,46.349,-69.353,172.333,26.924,154.941
C02848=1065.443,46.065,-69.333,172.331,26.921,154.940
C02849=1065.436,45.781,-69.315,172.329,26.917,154.940
C02850=1065.430,45.532,-69.299,172.327,26.915,154.940
C02851=1065.425,45.282,-69.282,172.326,26.912,154.939
C02852=1065.419,45.033,-69.266,172.325,26.910,154.939
C02853=1065.413,44.784,-69.250,172.324,26.907,154.938
C02854=1065.407,44.534,-69.233,172.323,26.904,154.938
C02855=1065.401,44.285,-69.217,172.321,26.901,154.937
C02856=1065.395,44.035,-69.200,172.320,26.899,154.937
C02857=1065.390,43.786,-69.184,172.318,26.896,154.937
C02858=1065.384,43.537,-69.168,172.317,26.893,154.936
C02859=1065.378,43.287,-69.152,172.315,26.890,154.936
C02860=1065.372,43.038,-69.135,172.314,26.888,154.936
C02861=1065.366,42.789,-69.119,172.312,26.885,154.935
C02862=1065.360,42.539,-69.103,172.311,26.882,154.935
C02863=1065.354,42.290,-69.087,172.309,26.879,154.935
C02864=1065.348,42.041,-69.070,172.309,26.877,154.934
C02865=1065.342,41.791,-69.054,172.307,26.875,154.934
C02866=1065.336,41.542,-69.038,172.306,26.872,154.933
C02867=1065.330,41.293,-69.022,172.304,26.869,154.933
C02868=1065.324,41.043,-69.005,172.303,26.867,154.933
C02869=1065.318,40.794,-68.989,172.301,26.864,154.932
C02870=1065.312,40.545,-68.973,172.300,26.861,154.932
C02871=1065.306,40.295,-68.957,172.298,26.859,154.932
C02872=1065.300,40.046,-68.940,172.297,26.856,154.931
C02873=1065.294,39.797,-68.924,172.295,26.853,154.931
C02874=1065.289,39.547,-68.908,172.294,26.851,154.931
C02875=1065.283,39.297,-68.892,172.292,26.848,154.930
C02876=1065.277,39.048,-68.876,172.291,26.845,154.930
C02877=1065.271,38.798,-68.860,172.290,26.842,154.929
C02878=1065.265,38.549,-68.843,172.289,26.840,154.929
C02879=1065.259,38.300,-68.827,172.287,26.837,154.929
C02880=1065.253,38.050,-68.812,172.286,26.834,154.928
C02881=1065.247,37.801,-68.796,172.285,26.832,154.928
C02882=1065.241,37.551,-68.780,172.283,26.829,154.928
C02883=1065.235,37.302,-68.763,172.282,26.826,154.927
C02884=1065.229,37.053,-68.747,172.280,26.824,154.927
C02885=1065.223,36.803,-68.732,172.279,26.821,154.927
C02886=1065.216,36.554,-68.716,172.277,26.818,154.926
C02887=1065.210,36.304,-68.700,172.276,26.816,154.926
C02888=1065.204,36.055,-68.683,172.274,26.813,154.926
C02889=1065.199,35.805,-68.668,172.273,26.810,154.925
C02890=1065.192,35.556,-68.652,172.271,26.808,154.925
C02891=1065.186,35.307,-68.636,172.271,26.806,154.924
C02892=1065.180,35.057,-68.620,172.269,26.803,154.924
C02893=1065.175,34.807,-68.604,172.268,26.800,154.924
C02894=1065.168,34.558,-68.589,172.266,26.798,154.923
C02895=1065.162,34.309,-68.572,172.265,26.795,154.923
C02896=1065.156,34.059,-68.557,172.263,26.792,154.923
C02897=1065.150,33.810,-68.541,172.262,26.790,154.922
C02898=1065.144,33.561,-68.525,172.260,26.787,154.922
C02899=1065.138,33.311,-68.509,172.259,26.785,154.922
C02900=1065.133,33.062,-68.493,172.257,26.782,154.921
C02901=1065.127,32.813,-68.477,172.256,26.779,154.921
C02902=1065.120,32.563,-68.462,172.254,26.777,154.921
C02903=1065.114,32.314,-68.446,172.253,26.774,154.920
C02904=1065.108,32.064,-68.430,172.252,26.772,154.920
C02905=1065.103,31.814,-68.414,172.251,26.769,154.920
C02906=1065.096,31.565,-68.399,172.249,26.766,154.919
C02907=1065.090,31.316,-68.382,172.248,26.764,154.919
C02908=1065.085,31.066,-68.367,172.246,26.761,154.918
C02909=1065.079,30.817,-68.350,172.245,26.758,154.918
C02910=1065.072,30.533,-68.333,172.244,26.755,154.918
C02911=1065.065,30.249,-68.315,172.242,26.752,154.917
C02912=1065.058,29.966,-68.298,172.240,26.749,154.917
C02913=1065.051,29.682,-68.280,172.238,26.746,154.917
C02914=1065.045,29.433,-68.264,172.237,26.743,154.916
C02915=1065.040,29.183,-68.248,172.235,26.741,154.916
C02916=1065.034,28.933,-68.232,172.234,26.738,154.915
C02917=1065.028,28.684,-68.217,172.232,26.735,154.915
C02918=1065.022,28.435,-68.201,172.232,26.733,154.915
C02919=1065.015,28.185,-68.186,172.230,26.731,154.914
C02920=1065.009,27.936,-68.170,172.229,26.728,154.914
C02921=1065.004,27.686,-68.154,172.227,26.725,154.914
C02922=1064.997,27.437,-68.139,172.226,26.723,154.913
C02923=1064.992,27.187,-68.123,172.224,26.720,154.913
C02924=1064.985,26.938,-68.107,172.223,26.717,154.913
C02925=1064.980,26.689,-68.092,172.221,26.715,154.912
C02926=1064.973,26.439,-68.077,172.220,26.712,154.912
C02927=1064.967,26.190,-68.061,172.219,26.709,154.912
C02928=1064.961,25.940,-68.046,172.217,26.707,154.911
C02929=1064.955,25.691,-68.030,172.216,26.704,154.911
C02930=1064.949,25.441,-68.015,172.214,26.702,154.911
C02931=1064.943,25.192,-67.999,172.213,26.699,154.910
C02932=1064.937,24.943,-67.984,172.212,26.697,154.910
C02933=1064.931,24.693,-67.968,172.211,26.694,154.910
C02934=1064.925,24.444,-67.953,172.209,26.692,154.909
C02935=1064.919,24.194,-67.937,172.208,26.689,154.909
C02936=1064.912,23.945,-67.922,172.206,26.686,154.909
C02937=1064.907,23.695,-67.906,172.205,26.684,154.908
C02938=1064.901,23.446,-67.891,172.203,26.681,154.908
C02939=1064.895,23.196,-67.875,172.202,26.679,154.908
C02940=1064.889,22.947,-67.860,172.200,26.676,154.907
C02941=1064.883,22.697,-67.845,172.199,26.674,154.907
C02942=1064.877,22.448,-67.829,172.197,26.671,154.907
C02943=1064.871,22.199,-67.814,172.196,26.668,154.906
C02944=1064.865,21.949,-67.799,172.194,26.666,154.906
C02945=1064.859,21.699,-67.783,172.193,26.663,154.905
C02946=1064.853,21.451,-67.768,172.192,26.661,154.905
C02947=1064.847,21.201,-67.753,172.191,26.658,154.905
C02948=1064.841,20.951,-67.738,172.189,26.656,154.904
C02949=1064.835,20.702,-67.721,172.188,26.653,154.904
C02950=1064.829,20.452,-67.706,172.186,26.650,154.904
C02951=1064.824,20.203,-67.691,172.185,26.648,154.903
C02952=1064.817,19.953,-67.676,172.184,26.645,154.903
C02953=1064.811,19.704,-67.661,172.182,26.642,154.903
C02954=1064.805,19.454,-67.645,172.181,26.640,154.902
C02955=1064.799,19.205,-67.630,172.179,26.637,154.902
C02956=1064.793,18.955,-67.616,172.178,26.634,154.902
C02957=1064.787,18.706,-67.599,172.176,26.632,154.901
C02958=1064.780,18.456,-67.584,172.175,26.629,154.901
C02959=1064.775,18.207,-67.570,172.173,26.627,154.901
C02960=1064.769,17.957,-67.554,172.173,26.624,154.900
C02961=1064.763,17.708,-67.539,172.171,26.622,154.900
C02962=1064.756,17.458,-67.524,172.170,26.619,154.900
C02963=1064.751,17.209,-67.508,172.168,26.617,154.899
C02964=1064.745,16.960,-67.493,172.167,26.614,154.899
C02965=1064.738,16.710,-67.479,172.165,26.612,154.899
C02966=1064.733,16.461,-67.463,172.164,26.609,154.898
C02967=1064.727,16.211,-67.448,172.162,26.607,154.898
C02968=1064.720,15.962,-67.433,172.161,26.604,154.898
C02969=1064.715,15.712,-67.418,172.159,26.601,154.897
C02970=1064.709,15.463,-67.403,172.158,26.599,154.897
C02971=1064.702,15.214,-67.388,172.156,26.596,154.897
C02972=1064.697,14.964,-67.372,172.155,26.593,154.896
C02973=1064.691,14.715,-67.358,172.153,26.591,154.896
C02974=1064.683,14.432,-67.340,172.152,26.588,154.896
C02975=1064.677,14.150,-67.324,172.150,26.585,154.895
C02976=1064.671,13.867,-67.306,172.149,26.583,154.895
C02977=1064.663,13.584,-67.289,172.148,26.580,154.895
C02978=1064.657,13.335,-67.275,172.146,26.577,154.894
C02979=1064.651,13.086,-67.260,172.145,26.575,154.894
C02980=1064.645,12.836,-67.245,172.143,26.572,154.894
C02981=1064.638,12.586,-67.230,172.142,26.570,154.893
C02982=1064.632,12.338,-67.215,172.140,26.567,154.893
C02983=1064.626,12.088,-67.200,172.139,26.565,154.893
C02984=1064.620,11.838,-67.186,172.137,26.562,154.892
C02985=1064.614,11.589,-67.171,172.136,26.560,154.892
C02986=1064.608,11.339,-67.155,172.134,26.557,154.892
C02987=1064.602,11.090,-67.140,172.133,26.555,154.891
C02988=1064.596,10.841,-67.126,172.131,26.552,154.891
C02989=1064.590,10.591,-67.111,172.130,26.550,154.891
C02990=1064.583,10.341,-67.096,172.128,26.547,154.890
C02991=1064.578,10.092,-67.082,172.127,26.545,154.890
C02992=1064.571,9.842,-67.067,172.125,26.542,154.890
C02993=1064.565,9.592,-67.052,172.125,26.540,154.889
C02994=1064.559,9.344,-67.038,172.123,26.537,154.889
C02995=1064.553,9.094,-67.023,172.122,26.535,154.889
C02996=1064.547,8.844,-67.008,172.120,26.532,154.888
C02997=1064.541,8.595,-66.993,172.119,26.530,154.888
C02998=1064.534,8.346,-66.978,172.117,26.527,154.888
C02999=1064.529,8.096,-66.963,172.116,26.525,154.888
C03000=1064.523,7.846,-66.949,172.114,26.523,154.887
C03001=1064.517,7.596,-66.934,172.113,26.520,154.887
C03002=1064.511,7.347,-66.919,172.111,26.517,154.887
C03003=1064.505,7.098,-66.904,172.110,26.515,154.886
C03004=1064.498,6.848,-66.889,172.108,26.512,154.886
C03005=1064.493,6.599,-66.875,172.107,26.510,154.886
C03006=1064.486,6.349,-66.861,172.105,26.507,154.885
C03007=1064.481,6.100,-66.846,172.104,26.505,154.885
C03008=1064.474,5.850,-66.831,172.102,26.502,154.885
C03009=1064.468,5.601,-66.816,172.101,26.500,154.884
C03010=1064.462,5.352,-66.802,172.099,26.497,154.884
C03011=1064.456,5.101,-66.787,172.098,26.495,154.884
C03012=1064.450,4.852,-66.773,172.097,26.492,154.883
C03013=1064.444,4.603,-66.758,172.096,26.490,154.883
C03014=1064.438,4.354,-66.743,172.094,26.488,154.883
C03015=1064.432,4.104,-66.729,172.093,26.485,154.882
C03016=1064.426,3.855,-66.714,172.091,26.483,154.882
C03017=1064.420,3.605,-66.699,172.090,26.480,154.882
C03018=1064.414,3.356,-66.685,172.088,26.477,154.882
C03019=1064.408,3.106,-66.671,172.087,26.475,154.881
C03020=1064.402,2.856,-66.656,172.086,26.472,154.881
C03021=1064.396,2.607,-66.641,172.084,26.470,154.881
C03022=1064.390,2.357,-66.627,172.082,26.468,154.880
C03023=1064.384,2.108,-66.612,172.081,26.465,154.880
C03024=1064.378,1.858,-66.597,172.080,26.462,154.880
C03025=1064.372,1.609,-66.583,172.078,26.460,154.879
C03026=1064.366,1.359,-66.569,172.077,26.457,154.879
C03027=1064.360,1.110,-66.554,172.075,26.455,154.879
C03028=1064.354,0.860,-66.540,172.074,26.452,154.878
C03029=1064.348,0.611,-66.525,172.072,26.450,154.878
C03030=1064.342,0.362,-66.511,172.071,26.447,154.878
C03031=1064.336,0.112,-66.496,172.069,26.445,154.877
C03032=1064.330,-0.137,-66.482,172.069,26.443,154.877
C03033=1064.324,-0.388,-66.468,172.067,26.440,154.877
C03034=1064.319,-0.637,-66.453,172.066,26.437,154.876
C03035=1064.312,-0.886,-66.438,172.064,26.435,154.876
C03036=1064.307,-1.136,-66.424,172.063,26.433,154.876
C03037=1064.300,-1.386,-66.409,172.061,26.430,154.876
C03038=1064.294,-1.666,-66.394,172.060,26.428,154.875
C03039=1064.287,-1.946,-66.377,172.057,26.424,154.875
C03040=1064.281,-2.226,-66.361,172.056,26.421,154.875
C03041=1064.274,-2.508,-66.345,172.055,26.419,154.874
C03042=1064.268,-2.757,-66.330,172.053,26.416,154.874
C03043=1064.262,-3.007,-66.316,172.051,26.414,154.874
C03044=1064.256,-3.256,-66.302,172.050,26.411,154.873
C03045=1064.250,-3.506,-66.288,172.049,26.409,154.873
C03046=1064.244,-3.755,-66.273,172.047,26.407,154.873
C03047=1064.238,-4.005,-66.259,172.046,26.404,154.872
C03048=1064.232,-4.254,-66.245,172.044,26.402,154.872
C03049=1064.225,-4.504,-66.231,172.043,26.399,154.872
C03050=1064.219,-4.753,-66.216,172.041,26.397,154.871
C03051=1064.213,-5.003,-66.202,172.040,26.394,154.871
C03052=1064.207,-5.252,-66.188,172.038,26.392,154.871
C03053=1064.201,-5.501,-66.174,172.036,26.390,154.871
C03054=1064.195,-5.752,-66.160,172.035,26.387,154.870
C03055=1064.189,-6.000,-66.146,172.035,26.385,154.870
C03056=1064.183,-6.251,-66.132,172.033,26.383,154.870
C03057=1064.177,-6.499,-66.117,172.031,26.380,154.869
C03058=1064.170,-6.749,-66.104,172.030,26.378,154.869
C03059=1064.164,-6.999,-66.090,172.028,26.376,154.869
C03060=1064.159,-7.248,-66.075,172.027,26.373,154.869
C03061=1064.152,-7.498,-66.061,172.026,26.370,154.868
C03062=1064.146,-7.747,-66.047,172.024,26.368,154.868
C03063=1064.140,-7.997,-66.033,172.022,26.366,154.868
C03064=1064.134,-8.246,-66.019,172.021,26.364,154.867
C03065=1064.127,-8.496,-66.004,172.019,26.361,154.867
C03066=1064.122,-8.746,-65.991,172.018,26.359,154.867
C03067=1064.116,-8.995,-65.977,172.017,26.356,154.867
C03068=1064.109,-9.245,-65.962,172.015,26.354,154.866
C03069=1064.104,-9.494,-65.949,172.013,26.351,154.866
C03070=1064.098,-9.743,-65.935,172.012,26.349,154.866
C03071=1064.091,-9.993,-65.920,172.010,26.347,154.865
C03072=1064.086,-10.243,-65.906,172.009,26.344,154.865
C03073=1064.079,-10.493,-65.893,172.008,26.342,154.865
C03074=1064.074,-10.742,-65.879,172.006,26.339,154.865
C03075=1064.067,-10.991,-65.865,172.004,26.337,154.864
C03076=1064.061,-11.241,-65.851,172.003,26.335,154.864
C03077=1064.055,-11.491,-65.837,172.001,26.332,154.864
C03078=1064.049,-11.740,-65.824,172.000,26.330,154.863
C03079=1064.043,-11.990,-65.809,171.998,26.328,154.863
C03080=1064.037,-12.239,-65.795,171.997,26.325,154.863
C03081=1064.031,-12.488,-65.782,171.996,26.322,154.863
C03082=1064.025,-12.739,-65.767,171.994,26.320,154.862
C03083=1064.019,-12.987,-65.753,171.992,26.318,154.862
C03084=1064.013,-13.237,-65.739,171.991,26.316,154.862
C03085=1064.008,-13.487,-65.726,171.989,26.313,154.861
C03086=1064.001,-13.737,-65.712,171.988,26.311,154.861
C03087=1063.995,-13.986,-65.698,171.986,26.309,154.861
C03088=1063.989,-14.235,-65.685,171.986,26.306,154.860
C03089=1063.983,-14.485,-65.670,171.984,26.304,154.860
C03090=1063.977,-14.735,-65.656,171.983,26.301,154.860
C03091=1063.971,-14.984,-65.643,171.981,26.299,154.860
C03092=1063.965,-15.234,-65.628,171.980,26.297,154.859
C03093=1063.959,-15.483,-65.615,171.978,26.294,154.859
C03094=1063.953,-15.733,-65.602,171.977,26.292,154.859
C03095=1063.947,-15.982,-65.588,171.975,26.290,154.859
C03096=1063.940,-16.232,-65.574,171.974,26.287,154.858
C03097=1063.935,-16.482,-65.561,171.972,26.285,154.858
C03098=1063.928,-16.730,-65.547,171.971,26.283,154.858
C03099=1063.921,-16.980,-65.533,171.969,26.281,154.858
C03100=1063.916,-17.230,-65.519,171.968,26.278,154.857
C03101=1063.910,-17.479,-65.506,171.966,26.276,154.857
C03102=1063.902,-17.759,-65.490,171.965,26.274,154.857
C03103=1063.896,-18.037,-65.475,171.962,26.271,154.856
C03104=1063.889,-18.316,-65.460,171.961,26.268,154.856
C03105=1063.882,-18.595,-65.445,171.959,26.266,154.856
C03106=1063.877,-18.844,-65.431,171.958,26.263,154.856
C03107=1063.870,-19.094,-65.417,171.956,26.261,154.855
C03108=1063.864,-19.344,-65.404,171.955,26.259,154.855
C03109=1063.858,-19.593,-65.390,171.953,26.256,154.855
C03110=1063.852,-19.843,-65.377,171.952,26.254,154.855
C03111=1063.846,-20.093,-65.363,171.950,26.252,154.854
C03112=1063.840,-20.342,-65.350,171.949,26.250,154.854
C03113=1063.833,-20.591,-65.336,171.947,26.247,154.854
C03114=1063.828,-20.841,-65.322,171.946,26.245,154.853
C03115=1063.822,-21.090,-65.309,171.944,26.243,154.853
C03116=1063.815,-21.341,-65.296,171.943,26.240,154.853
C03117=1063.810,-21.590,-65.282,171.941,26.238,154.853
C03118=1063.803,-21.840,-65.269,171.940,26.236,154.852
C03119=1063.797,-22.089,-65.256,171.938,26.233,154.852
C03120=1063.791,-22.339,-65.242,171.937,26.232,154.852
C03121=1063.785,-22.588,-65.228,171.935,26.229,154.852
C03122=1063.779,-22.838,-65.215,171.934,26.227,154.851
C03123=1063.773,-23.087,-65.201,171.932,26.225,154.851
C03124=1063.767,-23.337,-65.188,171.931,26.222,154.851
C03125=1063.761,-23.586,-65.175,171.929,26.220,154.851
C03126=1063.755,-23.837,-65.161,171.928,26.218,154.850
C03127=1063.749,-24.086,-65.148,171.926,26.215,154.850
C03128=1063.743,-24.335,-65.135,171.925,26.213,154.850
C03129=1063.737,-24.585,-65.121,171.923,26.211,154.850
C03130=1063.731,-24.834,-65.107,171.922,26.208,154.849
C03131=1063.725,-25.083,-65.094,171.920,26.206,154.849
C03132=1063.719,-25.334,-65.081,171.919,26.204,154.849
C03133=1063.713,-25.583,-65.067,171.917,26.201,154.848
C03134=1063.707,-25.833,-65.054,171.915,26.200,154.848
C03135=1063.701,-26.082,-65.040,171.914,26.197,154.848
C03136=1063.695,-26.332,-65.027,171.912,26.195,154.848
C03137=1063.689,-26.581,-65.014,171.911,26.193,154.848
C03138=1063.683,-26.831,-65.001,171.909,26.190,154.847
C03139=1063.676,-27.080,-64.988,171.908,26.188,154.847
C03140=1063.670,-27.330,-64.974,171.906,26.186,154.847
C03141=1063.664,-27.580,-64.961,171.905,26.184,154.847
C03142=1063.658,-27.829,-64.948,171.903,26.182,154.846
C03143=1063.652,-28.079,-64.935,171.902,26.179,154.846
C03144=1063.646,-28.328,-64.921,171.900,26.177,154.846
C03145=1063.640,-28.578,-64.909,171.899,26.175,154.846
C03146=1063.633,-28.828,-64.895,171.897,26.173,154.845
C03147=1063.627,-29.077,-64.882,171.896,26.171,154.845
C03148=1063.621,-29.327,-64.869,171.894,26.168,154.845
C03149=1063.615,-29.576,-64.856,171.893,26.166,154.845
C03150=1063.609,-29.826,-64.842,171.891,26.164,154.844
C03151=1063.603,-30.076,-64.830,171.889,26.162,154.844
C03152=1063.597,-30.325,-64.816,171.888,26.160,154.844
C03153=1063.591,-30.574,-64.803,171.886,26.157,154.844
C03154=1063.584,-30.825,-64.790,171.885,26.155,154.843
C03155=1063.578,-31.074,-64.777,171.883,26.153,154.843
C03156=1063.572,-31.323,-64.764,171.882,26.151,154.843
C03157=1063.566,-31.573,-64.751,171.880,26.149,154.843
C03158=1063.560,-31.822,-64.738,171.879,26.147,154.843
C03159=1063.554,-32.072,-64.725,171.877,26.144,154.842
C03160=1063.548,-32.322,-64.712,171.876,26.142,154.842
C03161=1063.542,-32.571,-64.699,171.874,26.140,154.842
C03162=1063.536,-32.821,-64.686,171.873,26.138,154.842
C03163=1063.529,-33.070,-64.673,171.871,26.136,154.841
C03164=1063.524,-33.320,-64.660,171.870,26.133,154.841
C03165=1063.517,-33.569,-64.647,171.868,26.132,154.841
C03166=1063.511,-33.848,-64.632,171.866,26.129,154.841
C03167=1063.504,-34.126,-64.618,171.865,26.127,154.840
C03168=1063.497,-34.404,-64.603,171.862,26.124,154.840
C03169=1063.490,-34.682,-64.588,171.861,26.122,154.840
C03170=1063.484,-34.932,-64.576,171.859,26.120,154.840
C03171=1063.478,-35.181,-64.563,171.858,26.117,154.839
C03172=1063.472,-35.431,-64.550,171.856,26.116,154.839
C03173=1063.466,-35.680,-64.537,171.855,26.113,154.839
C03174=1063.460,-35.930,-64.524,171.853,26.111,154.839
C03175=1063.454,-36.180,-64.512,171.852,26.109,154.838
C03176=1063.448,-36.429,-64.498,171.850,26.107,154.838
C03177=1063.442,-36.679,-64.486,171.849,26.105,154.838
C03178=1063.436,-36.929,-64.473,171.847,26.102,154.838
C03179=1063.430,-37.178,-64.460,171.846,26.100,154.838
C03180=1063.423,-37.428,-64.447,171.844,26.098,154.837
C03181=1063.418,-37.678,-64.434,171.843,26.096,154.837
C03182=1063.411,-37.927,-64.421,171.841,26.094,154.837
C03183=1063.406,-38.176,-64.409,171.839,26.092,154.837
C03184=1063.400,-38.426,-64.396,171.838,26.089,154.836
C03185=1063.394,-38.675,-64.383,171.836,26.088,154.836
C03186=1063.388,-38.925,-64.370,171.835,26.085,154.836
C03187=1063.382,-39.174,-64.357,171.833,26.084,154.836
C03188=1063.375,-39.424,-64.345,171.832,26.081,154.836
C03189=1063.369,-39.674,-64.333,171.830,26.080,154.835
C03190=1063.363,-39.923,-64.319,171.829,26.077,154.835
C03191=1063.357,-40.173,-64.307,171.827,26.075,154.835
C03192=1063.351,-40.423,-64.294,171.825,26.073,154.835
C03193=1063.344,-40.672,-64.282,171.824,26.071,154.835
C03194=1063.338,-40.922,-64.269,171.822,26.069,154.834
C03195=1063.332,-41.171,-64.256,171.821,26.067,154.834
C03196=1063.326,-41.421,-64.243,171.819,26.065,154.834
C03197=1063.320,-41.671,-64.231,171.818,26.063,154.834
C03198=1063.314,-41.920,-64.219,171.816,26.061,154.834
C03199=1063.308,-42.170,-64.206,171.814,26.059,154.833
C03200=1063.302,-42.419,-64.193,171.813,26.057,154.833
C03201=1063.296,-42.669,-64.180,171.811,26.055,154.833
C03202=1063.289,-42.919,-64.168,171.810,26.053,154.833
C03203=1063.283,-43.169,-64.156,171.808,26.051,154.833
C03204=1063.277,-43.418,-64.143,171.807,26.049,154.832
C03205=1063.271,-43.668,-64.130,171.805,26.047,154.832
C03206=1063.265,-43.918,-64.117,171.804,26.044,154.832
C03207=1063.258,-44.167,-64.105,171.802,26.043,154.832
C03208=1063.252,-44.417,-64.092,171.801,26.040,154.832
C03209=1063.247,-44.666,-64.080,171.798,26.038,154.831
C03210=1063.241,-44.916,-64.067,171.796,26.036,154.831
C03211=1063.234,-45.165,-64.056,171.795,26.034,154.831
C03212=1063.228,-45.415,-64.043,171.793,26.032,154.831
C03213=1063.222,-45.664,-64.030,171.792,26.030,154.831
C03214=1063.216,-45.914,-64.018,171.790,26.028,154.830
C03215=1063.210,-46.164,-64.005,171.789,26.026,154.830
C03216=1063.204,-46.414,-63.993,171.787,26.024,154.830
C03217=1063.198,-46.664,-63.980,171.786,26.022,154.830
C03218=1063.192,-46.912,-63.968,171.784,26.020,154.830
C03219=1063.186,-47.162,-63.956,171.782,26.018,154.829
C03220=1063.180,-47.412,-63.943,171.781,26.016,154.829
C03221=1063.174,-47.661,-63.930,171.779,26.014,154.829
C03222=1063.167,-47.911,-63.918,171.778,26.012,154.829
C03223=1063.161,-48.161,-63.906,171.776,26.010,154.829
C03224=1063.156,-48.410,-63.893,171.775,26.008,154.828
C03225=1063.149,-48.660,-63.881,171.773,26.006,154.828
C03226=1063.143,-48.910,-63.869,171.771,26.004,154.828
C03227=1063.137,-49.159,-63.856,171.770,26.002,154.828
C03228=1063.131,-49.409,-63.844,171.768,26.000,154.828
C03229=1063.125,-49.659,-63.832,171.767,25.998,154.827
C03230=1063.118,-49.937,-63.818,171.765,25.996,154.827
C03231=1063.111,-50.215,-63.804,171.763,25.994,154.827
C03232=1063.104,-50.494,-63.790,171.761,25.991,154.827
C03233=1063.098,-50.772,-63.777,171.760,25.990,154.827
C03234=1063.092,-51.022,-63.764,171.758,25.988,154.827
C03235=1063.085,-51.272,-63.752,171.756,25.985,154.826
C03236=1063.079,-51.522,-63.740,171.755,25.984,154.826
C03237=1063.073,-51.771,-63.728,171.753,25.982,154.826
C03238=1063.066,-52.020,-63.716,171.752,25.980,154.826
C03239=1063.060,-52.270,-63.704,171.750,25.978,154.826
C03240=1063.054,-52.520,-63.692,171.749,25.976,154.825
C03241=1063.048,-52.769,-63.679,171.747,25.974,154.825
C03242=1063.041,-53.019,-63.667,171.745,25.973,154.825
C03243=1063.035,-53.269,-63.656,171.744,25.971,154.825
C03244=1063.030,-53.518,-63.644,171.741,25.969,154.825
C03245=1063.023,-53.768,-63.632,171.740,25.967,154.825
C03246=1063.017,-54.018,-63.619,171.738,25.965,154.825
C03247=1063.010,-54.267,-63.607,171.736,25.963,154.824
C03248=1063.004,-54.517,-63.595,171.735,25.961,154.824
C03249=1062.998,-54.766,-63.583,171.733,25.959,154.824
C03250=1062.992,-55.016,-63.571,171.732,25.958,154.824
C03251=1062.986,-55.266,-63.559,171.730,25.956,154.824
C03252=1062.980,-55.516,-63.547,171.728,25.954,154.824
C03253=1062.973,-55.765,-63.536,171.727,25.952,154.823
C03254=1062.968,-56.015,-63.523,171.725,25.950,154.823
C03255=1062.961,-56.264,-63.511,171.724,25.948,154.823
C03256=1062.954,-56.514,-63.499,171.722,25.946,154.823
C03257=1062.948,-56.764,-63.487,171.720,25.945,154.823
C03258=1062.942,-57.014,-63.476,171.719,25.943,154.823
C03259=1062.936,-57.263,-63.464,171.717,25.941,154.823
C03260=1062.930,-57.513,-63.451,171.716,25.939,154.822
C03261=1062.923,-57.762,-63.440,171.714,25.937,154.822
C03262=1062.917,-58.012,-63.428,171.712,25.935,154.822
C03263=1062.912,-58.262,-63.416,171.711,25.934,154.822
C03264=1062.905,-58.511,-63.404,171.709,25.932,154.822
C03265=1062.899,-58.761,-63.392,171.708,25.930,154.822
C03266=1062.893,-59.011,-63.380,171.706,25.928,154.821
C03267=1062.887,-59.260,-63.369,171.704,25.927,154.821
C03268=1062.881,-59.510,-63.356,171.703,25.925,154.821
C03269=1062.874,-59.759,-63.344,171.700,25.923,154.821
C03270=1062.868,-60.008,-63.333,171.699,25.921,154.821
C03271=1062.862,-60.259,-63.321,171.697,25.919,154.821
C03272=1062.856,-60.508,-63.309,171.695,25.917,154.821
C03273=1062.850,-60.757,-63.297,171.694,25.916,154.820
C03274=1062.844,-61.008,-63.286,171.692,25.914,154.820
C03275=1062.838,-61.257,-63.273,171.691,25.912,154.820
C03276=1062.831,-61.507,-63.261,171.689,25.910,154.820
C03277=1062.825,-61.756,-63.250,171.687,25.908,154.820
C03278=1062.819,-62.006,-63.238,171.686,25.906,154.820
C03279=1062.813,-62.256,-63.226,171.684,25.904,154.819
C03280=1062.807,-62.505,-63.215,171.683,25.903,154.819
C03281=1062.801,-62.755,-63.203,171.681,25.901,154.819
C03282=1062.794,-63.005,-63.191,171.679,25.899,154.819
C03283=1062.789,-63.254,-63.180,171.678,25.897,154.819
C03284=1062.782,-63.504,-63.168,171.676,25.896,154.819
C03285=1062.777,-63.753,-63.156,171.675,25.894,154.819
C03286=1062.770,-64.003,-63.144,171.673,25.892,154.818
C03287=1062.764,-64.253,-63.132,171.671,25.890,154.818
C03288=1062.759,-64.503,-63.121,171.670,25.889,154.818
C03289=1062.752,-64.752,-63.109,171.668,25.887,154.818
C03290=1062.746,-65.002,-63.097,171.666,25.885,154.818
C03291=1062.740,-65.251,-63.086,171.665,25.883,154.818
C03292=1062.734,-65.501,-63.074,171.662,25.881,154.818
C03293=1062.728,-65.751,-63.063,171.661,25.879,154.818
C03294=1062.721,-66.030,-63.050,171.659,25.878,154.817
C03295=1062.714,-66.310,-63.037,171.658,25.876,154.817
C03296=1062.707,-66.590,-63.023,171.656,25.874,154.817
C03297=1062.701,-66.869,-63.010,171.653,25.872,154.817
C03298=1062.694,-67.120,-62.999,171.652,25.870,154.817
C03299=1062.688,-67.369,-62.987,171.650,25.869,154.817
C03300=1062.683,-67.619,-62.976,171.649,25.867,154.817
C03301=1062.676,-67.869,-62.964,171.647,25.865,154.816
C03302=1062.670,-68.118,-62.953,171.645,25.863,154.816
C03303=1062.665,-68.369,-62.941,171.644,25.862,154.816
C03304=1062.659,-68.617,-62.929,171.642,25.860,154.816
C03305=1062.652,-68.868,-62.918,171.640,25.858,154.816
C03306=1062.646,-69.116,-62.907,171.639,25.856,154.816
C03307=1062.641,-69.367,-62.895,171.637,25.854,154.816
C03308=1062.634,-69.616,-62.883,171.636,25.853,154.815
C03309=1062.628,-69.866,-62.872,171.634,25.852,154.815
C03310=1062.622,-70.115,-62.860,171.632,25.850,154.815
C03311=1062.616,-70.365,-62.849,171.631,25.848,154.815
C03312=1062.611,-70.615,-62.838,171.629,25.846,154.815
C03313=1062.604,-70.864,-62.826,171.627,25.844,154.815
C03314=1062.598,-71.114,-62.815,171.625,25.842,154.815
C03315=1062.592,-71.364,-62.803,171.623,25.841,154.815
C03316=1062.587,-71.613,-62.791,171.622,25.839,154.815
C03317=1062.580,-71.864,-62.780,171.620,25.838,154.814
C03318=1062.574,-72.112,-62.769,171.618,25.836,154.814
C03319=1062.568,-72.363,-62.757,171.617,25.834,154.814
C03320=1062.562,-72.612,-62.746,171.615,25.832,154.814
C03321=1062.556,-72.862,-62.734,171.614,25.831,154.814
C03322=1062.551,-73.111,-62.723,171.612,25.829,154.814
C03323=1062.544,-73.362,-62.712,171.610,25.827,154.814
C03324=1062.538,-73.610,-62.700,171.609,25.826,154.814
C03325=1062.532,-73.861,-62.689,171.607,25.824,154.813
C03326=1062.526,-74.110,-62.678,171.605,25.822,154.813
C03327=1062.520,-74.360,-62.667,171.604,25.821,154.813
C03328=1062.514,-74.609,-62.655,171.602,25.819,154.813
C03329=1062.507,-74.859,-62.644,171.600,25.818,154.813
C03330=1062.502,-75.109,-62.633,171.599,25.816,154.813
C03331=1062.495,-75.358,-62.621,171.597,25.815,154.813
C03332=1062.489,-75.608,-62.610,171.595,25.813,154.813
C03333=1062.483,-75.858,-62.599,171.594,25.811,154.813
C03334=1062.477,-76.108,-62.588,171.591,25.810,154.813
C03335=1062.471,-76.357,-62.577,171.590,25.808,154.812
C03336=1062.465,-76.607,-62.565,171.588,25.806,154.812
C03337=1062.459,-76.856,-62.554,171.586,25.805,154.812
C03338=1062.453,-77.106,-62.543,171.585,25.803,154.812
C03339=1062.447,-77.356,-62.532,171.583,25.802,154.812
C03340=1062.441,-77.606,-62.521,171.581,25.800,154.812
C03341=1062.435,-77.855,-62.509,171.580,25.798,154.812
C03342=1062.428,-78.105,-62.498,171.578,25.797,154.812
C03343=1062.423,-78.355,-62.487,171.576,25.795,154.812
C03344=1062.416,-78.604,-62.477,171.575,25.794,154.812
C03345=1062.410,-78.854,-62.466,171.573,25.792,154.812
C03346=1062.404,-79.103,-62.455,171.571,25.791,154.811
C03347=1062.398,-79.354,-62.444,171.570,25.790,154.811
C03348=1062.392,-79.603,-62.432,171.568,25.788,154.811
C03349=1062.385,-79.853,-62.421,171.566,25.787,154.811
C03350=1062.380,-80.102,-62.410,171.565,25.785,154.811
C03351=1062.373,-80.352,-62.399,171.563,25.784,154.811
C03352=1062.367,-80.602,-62.388,171.561,25.782,154.811
C03353=1062.361,-80.851,-62.378,171.559,25.780,154.811
C03354=1062.355,-81.101,-62.366,171.557,25.779,154.811
C03355=1062.348,-81.350,-62.356,171.555,25.777,154.811
C03356=1062.342,-81.601,-62.345,171.554,25.776,154.811
C03357=1062.336,-81.850,-62.334,171.552,25.774,154.811
C03358=1062.329,-82.133,-62.321,171.550,25.773,154.811
C03359=1062.322,-82.414,-62.309,171.549,25.771,154.810
C03360=1062.315,-82.696,-62.297,171.546,25.769,154.810
C03361=1062.308,-82.978,-62.284,171.544,25.768,154.810
C03362=1062.302,-83.228,-62.274,171.543,25.766,154.810
C03363=1062.295,-83.478,-62.263,171.541,25.765,154.810
C03364=1062.290,-83.727,-62.252,171.539,25.764,154.810
C03365=1062.283,-83.977,-62.242,171.538,25.762,154.810
C03366=1062.277,-84.227,-62.230,171.536,25.761,154.810
C03367=1062.271,-84.476,-62.220,171.534,25.760,154.810
C03368=1062.264,-84.726,-62.209,171.533,25.758,154.810
C03369=1062.258,-84.976,-62.198,171.530,25.757,154.810
C03370=1062.252,-85.225,-62.187,171.528,25.755,154.810
C03371=1062.245,-85.475,-62.177,171.527,25.754,154.810
C03372=1062.240,-85.724,-62.166,171.525,25.752,154.810
C03373=1062.234,-85.974,-62.155,171.523,25.751,154.810
C03374=1062.228,-86.224,-62.144,171.522,25.750,154.810
C03375=1062.221,-86.473,-62.133,171.520,25.748,154.810
C03376=1062.216,-86.723,-62.123,171.518,25.747,154.809
C03377=1062.209,-86.974,-62.112,171.517,25.745,154.809
C03378=1062.203,-87.223,-62.102,171.515,25.744,154.809
C03379=1062.197,-87.472,-62.091,171.513,25.743,154.809
C03380=1062.191,-87.722,-62.079,171.512,25.741,154.809
C03381=1062.184,-87.972,-62.069,171.510,25.740,154.809
C03382=1062.178,-88.221,-62.058,171.508,25.739,154.809
C03383=1062.171,-88.471,-62.048,171.506,25.737,154.809
C03384=1062.166,-88.721,-62.037,171.505,25.736,154.809
C03385=1062.160,-88.971,-62.027,171.503,25.735,154.809
C03386=1062.153,-89.220,-62.016,171.501,25.734,154.809
C03387=1062.147,-89.470,-62.005,171.499,25.731,154.809
C03388=1062.142,-89.719,-61.994,171.497,25.730,154.809
C03389=1062.135,-89.969,-61.985,171.495,25.729,154.809
C03390=1062.129,-90.219,-61.973,171.494,25.728,154.809
C03391=1062.123,-90.469,-61.963,171.492,25.726,154.809
C03392=1062.117,-90.718,-61.952,171.490,25.725,154.809
C03393=1062.111,-90.968,-61.941,171.488,25.724,154.809
C03394=1062.104,-91.218,-61.931,171.487,25.723,154.809
C03395=1062.099,-91.468,-61.921,171.485,25.721,154.808
C03396=1062.093,-91.717,-61.910,171.483,25.720,154.808
C03397=1062.086,-91.966,-61.899,171.482,25.718,154.808
C03398=1062.080,-92.217,-61.889,171.480,25.717,154.808
C03399=1062.075,-92.467,-61.878,171.478,25.716,154.808
C03400=1062.068,-92.716,-61.868,171.477,25.714,154.808
C03401=1062.063,-92.966,-61.858,171.475,25.713,154.808
C03402=1062.056,-93.216,-61.847,171.473,25.712,154.808
C03403=1062.050,-93.465,-61.836,171.471,25.711,154.808
C03404=1062.044,-93.715,-61.825,171.470,25.709,154.808
C03405=1062.038,-93.965,-61.816,171.468,25.708,154.808
C03406=1062.032,-94.214,-61.805,171.465,25.706,154.808
C03407=1062.025,-94.464,-61.794,171.464,25.705,154.808
C03408=1062.020,-94.714,-61.784,171.462,25.704,154.808
C03409=1062.013,-94.963,-61.774,171.460,25.703,154.808
C03410=1062.008,-95.213,-61.763,171.459,25.701,154.808
C03411=1062.002,-95.463,-61.753,171.457,25.700,154.808
C03412=1061.995,-95.713,-61.742,171.455,25.699,154.808
C03413=1061.990,-95.963,-61.732,171.453,25.697,154.808
C03414=1061.983,-96.212,-61.721,171.452,25.696,154.808
C03415=1061.977,-96.461,-61.711,171.450,25.695,154.808
C03416=1061.971,-96.711,-61.701,171.448,25.694,154.808
C03417=1061.966,-96.961,-61.690,171.447,25.692,154.808
C03418=1061.960,-97.211,-61.680,171.445,25.691,154.808
C03419=1061.953,-97.461,-61.669,171.443,25.690,154.808
C03420=1061.947,-97.710,-61.658,171.441,25.689,154.808
C03421=1061.941,-97.960,-61.649,171.440,25.688,154.808
C03422=1061.934,-98.244,-61.638,171.437,25.686,154.808
C03423=1061.927,-98.529,-61.626,171.435,25.685,154.808
C03424=1061.920,-98.813,-61.615,171.433,25.684,154.808
C03425=1061.913,-99.097,-61.603,171.431,25.682,154.808
C03426=1061.907,-99.346,-61.592,171.429,25.681,154.808
C03427=1061.900,-99.597,-61.581,171.427,25.680,154.808
C03428=1061.894,-99.846,-61.572,171.426,25.679,154.808
C03429=1061.888,-100.096,-61.561,171.424,25.678,154.808
C03430=1061.882,-100.346,-61.551,171.422,25.676,154.808
C03431=1061.876,-100.595,-61.542,171.420,25.675,154.808
C03432=1061.870,-100.845,-61.531,171.419,25.674,154.808
C03433=1061.864,-101.095,-61.521,171.417,25.673,154.808
C03434=1061.857,-101.345,-61.511,171.415,25.672,154.808
C03435=1061.851,-101.594,-61.501,171.413,25.671,154.808
C03436=1061.845,-101.844,-61.490,171.412,25.670,154.808
C03437=1061.839,-102.094,-61.480,171.410,25.669,154.808
C03438=1061.833,-102.343,-61.470,171.408,25.667,154.808
C03439=1061.827,-102.593,-61.460,171.406,25.666,154.808
C03440=1061.821,-102.843,-61.450,171.405,25.665,154.808
C03441=1061.815,-103.092,-61.440,171.402,25.664,154.808
C03442=1061.809,-103.343,-61.430,171.400,25.663,154.808
C03443=1061.802,-103.592,-61.419,171.399,25.662,154.808
C03444=1061.796,-103.842,-61.410,171.397,25.661,154.808
C03445=1061.790,-104.092,-61.400,171.395,25.659,154.808
C03446=1061.784,-104.341,-61.389,171.393,25.658,154.808
C03447=1061.778,-104.591,-61.380,171.391,25.658,154.808
C03448=1061.772,-104.841,-61.370,171.390,25.656,154.808
C03449=1061.766,-105.090,-61.359,171.388,25.655,154.808
C03450=1061.760,-105.340,-61.350,171.386,25.654,154.808
C03451=1061.754,-105.590,-61.340,171.385,25.653,154.808
C03452=1061.747,-105.839,-61.330,171.383,25.652,154.808
C03453=1061.742,-106.089,-61.320,171.381,25.651,154.808
C03454=1061.735,-106.339,-61.310,171.379,25.650,154.808
C03455=1061.729,-106.588,-61.300,171.377,25.649,154.808
C03456=1061.723,-106.838,-61.290,171.376,25.648,154.808
C03457=1061.717,-107.089,-61.280,171.374,25.647,154.808
C03458=1061.711,-107.338,-61.270,171.372,25.646,154.808
C03459=1061.704,-107.588,-61.260,171.370,25.645,154.808
C03460=1061.698,-107.837,-61.250,171.369,25.644,154.808
C03461=1061.692,-108.087,-61.241,171.366,25.642,154.808
C03462=1061.686,-108.337,-61.231,171.364,25.642,154.808
C03463=1061.679,-108.586,-61.221,171.362,25.640,154.808
C03464=1061.674,-108.836,-61.211,171.361,25.639,154.808
C03465=1061.668,-109.086,-61.201,171.359,25.639,154.808
C03466=1061.661,-109.336,-61.192,171.357,25.637,154.808
C03467=1061.655,-109.585,-61.181,171.355,25.637,154.808
C03468=1061.649,-109.835,-61.172,171.353,25.636,154.808
C03469=1061.643,-110.085,-61.162,171.352,25.634,154.808
C03470=1061.636,-110.334,-61.153,171.350,25.634,154.808
C03471=1061.630,-110.584,-61.143,171.348,25.633,154.808
C03472=1061.625,-110.834,-61.133,171.346,25.632,154.808
C03473=1061.618,-111.084,-61.123,171.345,25.631,154.808
C03474=1061.612,-111.333,-61.113,171.343,25.630,154.808
C03475=1061.606,-111.583,-61.104,171.341,25.629,154.808
C03476=1061.600,-111.833,-61.094,171.339,25.628,154.808
C03477=1061.594,-112.083,-61.084,171.337,25.627,154.808
C03478=1061.587,-112.333,-61.075,171.336,25.626,154.808
C03479=1061.581,-112.582,-61.065,171.334,25.625,154.809
C03480=1061.575,-112.831,-61.055,171.332,25.624,154.809
C03481=1061.569,-113.081,-61.045,171.330,25.624,154.809
C03482=1061.562,-113.331,-61.036,171.328,25.622,154.809
C03483=1061.556,-113.581,-61.026,171.326,25.622,154.809
C03484=1061.551,-113.831,-61.016,171.324,25.620,154.809
C03485=1061.545,-114.081,-61.007,171.322,25.620,154.809
C03486=1061.537,-114.363,-60.996,171.320,25.619,154.809
C03487=1061.531,-114.646,-60.985,171.319,25.618,154.809
C03488=1061.523,-114.928,-60.974,171.316,25.616,154.809
C03489=1061.517,-115.211,-60.964,171.314,25.616,154.809
C03490=1061.511,-115.461,-60.954,171.312,25.615,154.809
C03491=1061.505,-115.711,-60.944,171.310,25.614,154.809
C03492=1061.498,-115.961,-60.935,171.309,25.613,154.809
C03493=1061.492,-116.210,-60.925,171.307,25.612,154.809
C03494=1061.487,-116.460,-60.916,171.305,25.612,154.809
C03495=1061.481,-116.709,-60.907,171.303,25.610,154.809
C03496=1061.474,-116.959,-60.897,171.301,25.610,154.809
C03497=1061.468,-117.209,-60.887,171.300,25.609,154.810
C03498=1061.461,-117.458,-60.878,171.298,25.608,154.810
C03499=1061.455,-117.708,-60.869,171.296,25.607,154.810
C03500=1061.449,-117.958,-60.859,171.294,25.607,154.810
C03501=1061.443,-118.208,-60.850,171.292,25.606,154.810
C03502=1061.437,-118.458,-60.840,171.290,25.605,154.810
C03503=1061.430,-118.707,-60.831,171.288,25.604,154.810
C03504=1061.424,-118.957,-60.821,171.286,25.603,154.810
C03505=1061.419,-119.206,-60.812,171.284,25.602,154.810
C03506=1061.412,-119.456,-60.802,171.282,25.602,154.810
C03507=1061.406,-119.706,-60.793,171.281,25.600,154.810
C03508=1061.400,-119.956,-60.784,171.279,25.600,154.810
C03509=1061.394,-120.206,-60.774,171.277,25.599,154.810
C03510=1061.387,-120.456,-60.765,171.275,25.599,154.810
C03511=1061.381,-120.705,-60.756,171.273,25.597,154.810
C03512=1061.375,-120.955,-60.746,171.271,25.597,154.811
C03513=1061.369,-121.204,-60.737,171.270,25.596,154.811
C03514=1061.363,-121.454,-60.727,171.268,25.596,154.811
C03515=1061.357,-121.704,-60.718,171.266,25.594,154.811
C03516=1061.351,-121.954,-60.709,171.264,25.594,154.811
C03517=1061.344,-122.204,-60.700,171.262,25.593,154.811
C03518=1061.338,-122.454,-60.690,171.260,25.593,154.811
C03519=1061.332,-122.703,-60.681,171.258,25.592,154.811
C03520=1061.326,-122.952,-60.672,171.257,25.591,154.811
C03521=1061.321,-123.203,-60.663,171.255,25.590,154.811
C03522=1061.314,-123.453,-60.653,171.253,25.590,154.811
C03523=1061.308,-123.702,-60.644,171.251,25.589,154.811
C03524=1061.301,-123.952,-60.635,171.249,25.588,154.812
C03525=1061.296,-124.201,-60.626,171.247,25.588,154.812
C03526=1061.290,-124.451,-60.617,171.246,25.587,154.812
C03527=1061.284,-124.701,-60.607,171.244,25.586,154.812
C03528=1061.277,-124.951,-60.598,171.242,25.585,154.812
C03529=1061.271,-125.201,-60.589,171.240,25.585,154.812
C03530=1061.265,-125.451,-60.580,171.237,25.584,154.812
C03531=1061.259,-125.700,-60.571,171.236,25.583,154.812
C03532=1061.252,-125.950,-60.562,171.234,25.583,154.812
C03533=1061.246,-126.200,-60.553,171.232,25.582,154.812
C03534=1061.240,-126.450,-60.543,171.230,25.581,154.813
C03535=1061.234,-126.700,-60.534,171.228,25.581,154.813
C03536=1061.228,-126.948,-60.525,171.226,25.580,154.813
C03537=1061.222,-127.199,-60.516,171.224,25.580,154.813
C03538=1061.216,-127.449,-60.507,171.223,25.579,154.813
C03539=1061.209,-127.698,-60.498,171.221,25.578,154.813
C03540=1061.204,-127.948,-60.489,171.219,25.577,154.813
C03541=1061.199,-128.198,-60.478,171.217,25.576,154.813
C03542=1061.196,-128.449,-60.468,171.216,25.574,154.813
C03543=1061.195,-128.699,-60.457,171.214,25.572,154.813
C03544=1061.194,-128.950,-60.445,171.214,25.569,154.812
C03545=1061.196,-129.200,-60.431,171.213,25.565,154.812
C03546=1061.199,-129.453,-60.418,171.212,25.560,154.811
C03547=1061.203,-129.703,-60.403,171.211,25.555,154.810
C03548=1061.209,-129.954,-60.389,171.211,25.550,154.809
C03549=1061.216,-130.205,-60.373,171.210,25.544,154.808
C03550=1060.836,-130.227,-60.564,171.163,25.701,154.841
C03551=1060.829,-129.977,-60.580,171.163,25.707,154.842
C03552=1060.823,-129.726,-60.595,171.163,25.712,154.843
C03553=1060.819,-129.475,-60.610,171.164,25.717,154.844
C03554=1060.816,-129.223,-60.623,171.165,25.722,154.845
C03555=1060.815,-128.973,-60.636,171.165,25.725,154.845
C03556=1060.814,-128.722,-60.648,171.167,25.728,154.846
C03557=1060.816,-128.471,-60.660,171.168,25.731,154.846
C03558=1060.819,-128.221,-60.671,171.170,25.733,154.846
C03559=1060.823,-127.970,-60.680,171.171,25.734,154.846
C03560=1060.829,-127.721,-60.690,171.173,25.735,154.846
C03561=1060.835,-127.472,-60.699,171.175,25.735,154.846
C03562=1060.841,-127.221,-60.707,171.177,25.736,154.846
C03563=1060.847,-126.972,-60.717,171.179,25.737,154.846
C03564=1060.854,-126.722,-60.727,171.181,25.737,154.846
C03565=1060.859,-126.473,-60.736,171.182,25.738,154.846
C03566=1060.866,-126.223,-60.744,171.184,25.738,154.846
C03567=1060.872,-125.973,-60.754,171.186,25.739,154.845
C03568=1060.878,-125.723,-60.763,171.188,25.740,154.845
C03569=1060.885,-125.473,-60.771,171.190,25.740,154.845
C03570=1060.890,-125.224,-60.781,171.192,25.741,154.845
C03571=1060.896,-124.974,-60.790,171.194,25.742,154.845
C03572=1060.903,-124.724,-60.800,171.196,25.743,154.845
C03573=1060.909,-124.474,-60.808,171.198,25.744,154.845
C03574=1060.915,-124.224,-60.818,171.200,25.744,154.845
C03575=1060.922,-123.975,-60.827,171.202,25.745,154.845
C03576=1060.927,-123.725,-60.836,171.204,25.745,154.845
C03577=1060.933,-123.475,-60.845,171.206,25.746,154.844
C03578=1060.940,-123.226,-60.854,171.207,25.747,154.844
C03579=1060.946,-122.976,-60.864,171.209,25.748,154.844
C03580=1060.952,-122.726,-60.873,171.211,25.748,154.844
C03581=1060.958,-122.476,-60.883,171.213,25.749,154.844
C03582=1060.964,-122.226,-60.891,171.215,25.750,154.844
C03583=1060.970,-121.977,-60.901,171.217,25.750,154.844
C03584=1060.976,-121.727,-60.910,171.218,25.751,154.844
C03585=1060.983,-121.477,-60.919,171.220,25.752,154.844
C03586=1060.989,-121.228,-60.929,171.222,25.753,154.844
C03587=1060.995,-120.978,-60.939,171.224,25.753,154.844
C03588=1061.001,-120.728,-60.947,171.226,25.754,154.844
C03589=1061.007,-120.478,-60.957,171.228,25.755,154.844
C03590=1061.013,-120.228,-60.966,171.229,25.756,154.843
C03591=1061.019,-119.979,-60.976,171.231,25.756,154.843
C03592=1061.025,-119.729,-60.985,171.233,25.757,154.843
C03593=1061.031,-119.479,-60.995,171.235,25.758,154.843
C03594=1061.038,-119.230,-61.004,171.238,25.759,154.843
C03595=1061.045,-118.980,-61.013,171.240,25.759,154.843
C03596=1061.051,-118.730,-61.023,171.241,25.761,154.843
C03597=1061.056,-118.481,-61.032,171.243,25.761,154.843
C03598=1061.062,-118.231,-61.042,171.245,25.762,154.843
C03599=1061.068,-117.981,-61.051,171.247,25.763,154.843
C03600=1061.074,-117.731,-61.060,171.249,25.764,154.843
C03601=1061.081,-117.481,-61.070,171.250,25.764,154.843
C03602=1061.087,-117.231,-61.079,171.252,25.765,154.843
C03603=1061.093,-116.981,-61.089,171.254,25.766,154.843
C03604=1061.099,-116.732,-61.098,171.256,25.767,154.842
C03605=1061.105,-116.482,-61.108,171.258,25.768,154.842
C03606=1061.112,-116.232,-61.118,171.259,25.768,154.842
C03607=1061.118,-115.982,-61.127,171.261,25.770,154.842
C03608=1061.124,-115.732,-61.137,171.263,25.770,154.842
C03609=1061.129,-115.483,-61.146,171.265,25.771,154.842
C03610=1061.136,-115.234,-61.156,171.267,25.772,154.842
C03611=1061.144,-114.951,-61.167,171.269,25.773,154.842
C03612=1061.150,-114.668,-61.177,171.271,25.774,154.842
C03613=1061.158,-114.385,-61.188,171.273,25.775,154.842
C03614=1061.164,-114.102,-61.199,171.276,25.776,154.842
C03615=1061.170,-113.853,-61.209,171.278,25.777,154.842
C03616=1061.177,-113.603,-61.219,171.279,25.778,154.842
C03617=1061.183,-113.354,-61.228,171.281,25.779,154.842
C03618=1061.189,-113.104,-61.238,171.283,25.780,154.842
